C05459=1078.522,130.349,-70.098,174.153,23.499,154.054
C05460=1078.528,130.599,-70.117,174.156,23.501,154.054
C05461=1078.534,130.848,-70.137,174.158,23.504,154.054
C05462=1078.540,131.096,-70.157,174.159,23.506,154.055
C05463=1078.545,131.346,-70.177,174.162,23.509,154.055
C05464=1078.551,131.595,-70.197,174.163,23.510,154.055
C05465=1078.557,131.844,-70.217,174.165,23.513,154.055
C05466=1078.563,132.093,-70.236,174.167,23.515,154.056
C05467=1078.568,132.342,-70.257,174.169,23.517,154.056
C05468=1078.574,132.591,-70.277,174.170,23.520,154.056
C05469=1078.580,132.841,-70.296,174.173,23.522,154.056
C05470=1078.585,133.090,-70.317,174.174,23.524,154.056
C05471=1078.591,133.339,-70.337,174.176,23.527,154.057
C05472=1078.596,133.588,-70.357,174.178,23.529,154.057
C05473=1078.602,133.837,-70.376,174.180,23.532,154.057
C05474=1078.607,134.086,-70.397,174.181,23.533,154.057
C05475=1078.613,134.335,-70.417,174.184,23.536,154.058
C05476=1078.619,134.584,-70.437,174.186,23.538,154.058
C05477=1078.625,134.833,-70.457,174.187,23.541,154.058
C05478=1078.630,135.083,-70.478,174.190,23.543,154.058
C05479=1078.636,135.332,-70.498,174.191,23.545,154.058
C05480=1078.642,135.581,-70.518,174.193,23.548,154.058
C05481=1078.647,135.830,-70.538,174.195,23.550,154.059
C05482=1078.653,136.079,-70.558,174.197,23.552,154.059
C05483=1078.659,136.328,-70.579,174.198,23.555,154.059
C05484=1078.664,136.578,-70.598,174.201,23.557,154.059
C05485=1078.670,136.827,-70.618,174.203,23.559,154.059
C05486=1078.676,137.075,-70.638,174.204,23.561,154.060
C05487=1078.681,137.325,-70.659,174.207,23.564,154.060
C05488=1078.687,137.574,-70.679,174.208,23.566,154.060
C05489=1078.693,137.823,-70.700,174.210,23.568,154.060
C05490=1078.699,138.072,-70.720,174.212,23.571,154.061
C05491=1078.704,138.321,-70.740,174.214,23.573,154.061
C05492=1078.710,138.570,-70.760,174.215,23.575,154.061
C05493=1078.715,138.819,-70.781,174.218,23.577,154.061
C05494=1078.720,139.068,-70.801,174.220,23.580,154.061
C05495=1078.727,139.318,-70.822,174.221,23.582,154.062
C05496=1078.732,139.567,-70.842,174.224,23.584,154.062
C05497=1078.738,139.816,-70.862,174.225,23.587,154.062
C05498=1078.744,140.065,-70.883,174.228,23.589,154.062
C05499=1078.750,140.314,-70.903,174.229,23.591,154.063
C05500=1078.755,140.563,-70.923,174.231,23.594,154.063
C05501=1078.760,140.812,-70.944,174.233,23.596,154.063
C05502=1078.767,141.061,-70.964,174.235,23.598,154.063
C05503=1078.772,141.310,-70.985,174.237,23.601,154.063
C05504=1078.777,141.560,-71.005,174.239,23.603,154.064
C05505=1078.783,141.808,-71.025,174.241,23.605,154.064
C05506=1078.788,142.058,-71.046,174.243,23.608,154.064
C05507=1078.794,142.307,-71.066,174.244,23.610,154.064
C05508=1078.800,142.557,-71.087,174.247,23.612,154.064
C05509=1078.806,142.805,-71.107,174.248,23.615,154.065
C05510=1078.812,143.086,-71.131,174.251,23.617,154.065
C05511=1078.818,143.367,-71.154,174.253,23.620,154.065
C05512=1078.824,143.647,-71.176,174.255,23.622,154.065
C05513=1078.831,143.928,-71.200,174.257,23.625,154.066
C05514=1078.836,144.177,-71.221,174.260,23.627,154.066
C05515=1078.842,144.427,-71.242,174.261,23.629,154.066
C05516=1078.848,144.675,-71.262,174.263,23.632,154.066
C05517=1078.853,144.925,-71.282,174.265,23.634,154.066
C05518=1078.859,145.173,-71.303,174.267,23.637,154.067
C05519=1078.864,145.422,-71.324,174.269,23.639,154.067
C05520=1078.871,145.672,-71.344,174.271,23.641,154.067
C05521=1078.876,145.921,-71.365,174.273,23.643,154.067
C05522=1078.881,146.169,-71.386,174.274,23.645,154.067
C05523=1078.887,146.418,-71.407,174.277,23.648,154.068
C05524=1078.893,146.668,-71.427,174.279,23.650,154.068
C05525=1078.898,146.917,-71.448,174.281,23.652,154.068
C05526=1078.904,147.166,-71.469,174.283,23.655,154.068
C05527=1078.910,147.415,-71.490,174.285,23.657,154.068
C05528=1078.916,147.664,-71.510,174.286,23.659,154.069
C05529=1078.921,147.913,-71.530,174.289,23.662,154.069
C05530=1078.927,148.162,-71.552,174.290,23.663,154.069
C05531=1078.933,148.412,-71.572,174.293,23.666,154.069
C05532=1078.938,148.661,-71.593,174.295,23.668,154.069
C05533=1078.943,148.909,-71.614,174.296,23.671,154.070
C05534=1078.949,149.158,-71.635,174.299,23.673,154.070
C05535=1078.955,149.408,-71.655,174.301,23.675,154.070
C05536=1078.961,149.656,-71.676,174.302,23.677,154.070
C05537=1078.966,149.906,-71.697,174.305,23.680,154.070
C05538=1078.972,150.155,-71.719,174.306,23.682,154.071
C05539=1078.977,150.404,-71.739,174.308,23.684,154.071
C05540=1078.983,150.653,-71.760,174.311,23.687,154.071
C05541=1078.989,150.902,-71.781,174.312,23.689,154.071
C05542=1078.994,151.151,-71.802,174.314,23.691,154.071
C05543=1079.000,151.400,-71.823,174.317,23.694,154.072
C05544=1079.005,151.649,-71.844,174.318,23.696,154.072
C05545=1079.011,151.898,-71.865,174.321,23.698,154.072
C05546=1079.016,152.147,-71.886,174.323,23.701,154.072
C05547=1079.022,152.396,-71.907,174.324,23.702,154.072
C05548=1079.028,152.646,-71.928,174.326,23.705,154.073
C05549=1079.033,152.894,-71.949,174.328,23.707,154.073
C05550=1079.039,153.143,-71.970,174.330,23.709,154.073
C05551=1079.045,153.392,-71.992,174.333,23.712,154.073
C05552=1079.050,153.642,-72.012,174.334,23.714,154.073
C05553=1079.056,153.890,-72.033,174.336,23.716,154.073
C05554=1079.061,154.140,-72.054,174.339,23.719,154.074
C05555=1079.067,154.388,-72.076,174.340,23.721,154.074
C05556=1079.073,154.638,-72.096,174.342,23.723,154.074
C05557=1079.078,154.887,-72.118,174.345,23.726,154.074
C05558=1079.084,155.135,-72.139,174.346,23.727,154.074
C05559=1079.090,155.385,-72.160,174.349,23.730,154.075
C05560=1079.095,155.634,-72.181,174.351,23.732,154.075
C05561=1079.101,155.883,-72.202,174.352,23.734,154.075
C05562=1079.107,156.132,-72.223,174.354,23.737,154.075
C05563=1079.112,156.380,-72.245,174.357,23.739,154.075
C05564=1079.117,156.631,-72.266,174.358,23.741,154.076
C05565=1079.123,156.879,-72.287,174.361,23.744,154.076
C05566=1079.129,157.128,-72.309,174.363,23.746,154.076
C05567=1079.134,157.377,-72.330,174.364,23.748,154.076
C05568=1079.140,157.626,-72.351,174.367,23.751,154.076
C05569=1079.146,157.875,-72.373,174.369,23.753,154.077
C05570=1079.151,158.124,-72.393,174.371,23.755,154.077
C05571=1079.157,158.374,-72.415,174.373,23.757,154.077
C05572=1079.162,158.622,-72.437,174.375,23.760,154.077
C05573=1079.168,158.871,-72.458,174.377,23.762,154.077
C05574=1079.175,159.152,-72.482,174.380,23.764,154.078
C05575=1079.181,159.432,-72.506,174.382,23.767,154.078
C05576=1079.187,159.712,-72.529,174.384,23.769,154.078
C05577=1079.193,159.993,-72.554,174.387,23.772,154.078
C05578=1079.199,160.242,-72.575,174.388,23.774,154.078
C05579=1079.205,160.491,-72.597,174.390,23.777,154.079
C05580=1079.211,160.740,-72.618,174.393,23.779,154.079
C05581=1079.216,160.989,-72.639,174.395,23.781,154.079
C05582=1079.222,161.238,-72.661,174.396,23.784,154.079
C05583=1079.227,161.487,-72.682,174.399,23.786,154.079
C05584=1079.233,161.736,-72.704,174.401,23.788,154.080
C05585=1079.238,161.985,-72.726,174.402,23.790,154.080
C05586=1079.244,162.234,-72.747,174.405,23.793,154.080
C05587=1079.249,162.483,-72.769,174.407,23.795,154.080
C05588=1079.255,162.732,-72.791,174.409,23.797,154.080
C05589=1079.260,162.982,-72.812,174.411,23.800,154.081
C05590=1079.265,163.230,-72.833,174.413,23.802,154.081
C05591=1079.271,163.480,-72.855,174.415,23.805,154.081
C05592=1079.276,163.728,-72.877,174.417,23.807,154.081
C05593=1079.282,163.977,-72.898,174.419,23.809,154.081
C05594=1079.287,164.226,-72.920,174.422,23.812,154.082
C05595=1079.293,164.475,-72.942,174.424,23.814,154.082
C05596=1079.298,164.724,-72.964,174.425,23.816,154.082
C05597=1079.304,164.973,-72.985,174.428,23.818,154.082
C05598=1079.309,165.222,-73.007,174.430,23.821,154.082
C05599=1079.315,165.471,-73.029,174.432,23.823,154.083
C05600=1079.320,165.721,-73.051,174.434,23.825,154.083
C05601=1079.326,165.969,-73.072,174.436,23.828,154.083
C05602=1079.331,166.219,-73.094,174.438,23.830,154.083
C05603=1079.337,166.467,-73.116,174.440,23.832,154.083
C05604=1079.342,166.717,-73.138,174.442,23.835,154.084
C05605=1079.347,166.965,-73.160,174.444,23.837,154.084
C05606=1079.353,167.215,-73.181,174.447,23.840,154.084
C05607=1079.358,167.463,-73.203,174.448,23.841,154.084
C05608=1079.364,167.712,-73.226,174.450,23.844,154.084
C05609=1079.369,167.961,-73.248,174.453,23.846,154.085
C05610=1079.375,168.210,-73.269,174.455,23.848,154.085
C05611=1079.380,168.459,-73.291,174.457,23.851,154.085
C05612=1079.386,168.708,-73.313,174.459,23.853,154.085
C05613=1079.391,168.957,-73.335,174.461,23.855,154.085
C05614=1079.397,169.206,-73.356,174.464,23.858,154.086
C05615=1079.403,169.456,-73.378,174.466,23.860,154.086
C05616=1079.408,169.704,-73.401,174.467,23.863,154.086
C05617=1079.414,169.953,-73.423,174.470,23.865,154.086
C05618=1079.419,170.202,-73.444,174.472,23.867,154.086
C05619=1079.425,170.451,-73.466,174.474,23.870,154.087
C05620=1079.431,170.700,-73.488,174.476,23.871,154.087
C05621=1079.436,170.948,-73.510,174.478,23.874,154.087
C05622=1079.442,171.198,-73.533,174.480,23.876,154.087
C05623=1079.447,171.447,-73.554,174.483,23.879,154.087
C05624=1079.453,171.696,-73.576,174.484,23.880,154.087
C05625=1079.459,171.945,-73.599,174.487,23.883,154.088
C05626=1079.464,172.193,-73.620,174.489,23.885,154.088
C05627=1079.470,172.443,-73.642,174.491,23.888,154.088
C05628=1079.475,172.691,-73.665,174.494,23.890,154.088
C05629=1079.481,172.940,-73.687,174.495,23.892,154.088
C05630=1079.486,173.190,-73.709,174.497,23.894,154.089
C05631=1079.491,173.438,-73.732,174.500,23.897,154.089
C05632=1079.498,173.687,-73.753,174.502,23.899,154.089
C05633=1079.503,173.937,-73.775,174.504,23.901,154.089
C05634=1079.509,174.185,-73.797,174.506,23.903,154.089
C05635=1079.514,174.434,-73.820,174.508,23.905,154.089
C05636=1079.520,174.684,-73.842,174.511,23.908,154.090
C05637=1079.526,174.932,-73.864,174.513,23.910,154.090
C05638=1079.532,175.212,-73.889,174.515,23.913,154.090
C05639=1079.538,175.492,-73.914,174.518,23.915,154.090
C05640=1079.545,175.773,-73.939,174.520,23.918,154.091
C05641=1079.551,176.053,-73.964,174.522,23.920,154.091
C05642=1079.557,176.302,-73.987,174.525,23.922,154.091
C05643=1079.562,176.550,-74.008,174.527,23.925,154.091
C05644=1079.568,176.800,-74.031,174.529,23.927,154.091
C05645=1079.573,177.049,-74.054,174.532,23.930,154.091
C05646=1079.579,177.298,-74.075,174.533,23.931,154.092
C05647=1079.585,177.546,-74.098,174.535,23.934,154.092
C05648=1079.590,177.795,-74.120,174.538,23.936,154.092
C05649=1079.597,178.044,-74.142,174.540,23.939,154.092
C05650=1079.602,178.293,-74.165,174.543,23.941,154.092
C05651=1079.607,178.542,-74.187,174.545,23.943,154.092
C05652=1079.614,178.790,-74.209,174.546,23.945,154.093
C05653=1079.619,179.040,-74.232,174.549,23.947,154.093
C05654=1079.625,179.289,-74.255,174.551,23.950,154.093
C05655=1079.630,179.538,-74.277,174.554,23.952,154.093
C05656=1079.636,179.786,-74.299,174.556,23.955,154.093
C05657=1079.642,180.035,-74.322,174.558,23.957,154.093
C05658=1079.647,180.285,-74.344,174.560,23.959,154.094
C05659=1079.654,180.533,-74.366,174.562,23.961,154.094
C05660=1079.659,180.783,-74.389,174.564,23.963,154.094
C05661=1079.665,181.032,-74.412,174.567,23.966,154.094
C05662=1079.670,181.280,-74.434,174.569,23.968,154.094
C05663=1079.676,181.529,-74.456,174.571,23.970,154.094
C05664=1079.682,181.778,-74.479,174.574,23.972,154.095
C05665=1079.688,182.027,-74.502,174.575,23.974,154.095
C05666=1079.693,182.276,-74.524,174.578,23.976,154.095
C05667=1079.699,182.525,-74.546,174.580,23.979,154.095
C05668=1079.705,182.774,-74.569,174.582,23.981,154.095
C05669=1079.710,183.022,-74.592,174.585,23.983,154.095
C05670=1079.716,183.271,-74.614,174.587,23.986,154.096
C05671=1079.721,183.520,-74.637,174.590,23.988,154.096
C05672=1079.728,183.769,-74.659,174.592,23.990,154.096
C05673=1079.734,184.018,-74.682,174.594,23.992,154.096
C05674=1079.739,184.267,-74.704,174.596,23.995,154.096
C05675=1079.745,184.516,-74.727,174.598,23.997,154.096
C05676=1079.751,184.765,-74.750,174.601,23.999,154.097
C05677=1079.757,185.014,-74.773,174.603,24.001,154.097
C05678=1079.763,185.263,-74.796,174.605,24.003,154.097
C05679=1079.767,185.511,-74.819,174.608,24.006,154.097
C05680=1079.773,185.761,-74.841,174.610,24.008,154.097
C05681=1079.778,186.010,-74.864,174.611,24.011,154.098
C05682=1079.784,186.258,-74.887,174.614,24.013,154.098
C05683=1079.790,186.507,-74.910,174.616,24.015,154.098
C05684=1079.795,186.756,-74.932,174.618,24.018,154.098
C05685=1079.800,187.005,-74.956,174.621,24.020,154.098
C05686=1079.806,187.254,-74.979,174.623,24.023,154.099
C05687=1079.811,187.503,-75.002,174.625,24.025,154.099
C05688=1079.817,187.751,-75.025,174.628,24.027,154.099
C05689=1079.823,188.000,-75.048,174.630,24.030,154.099
C05690=1079.827,188.249,-75.071,174.633,24.032,154.099
C05691=1079.833,188.498,-75.094,174.634,24.034,154.099
C05692=1079.839,188.747,-75.117,174.636,24.036,154.100
C05693=1079.844,188.996,-75.140,174.639,24.039,154.100
C05694=1079.850,189.244,-75.163,174.641,24.041,154.100
C05695=1079.855,189.494,-75.186,174.643,24.044,154.100
C05696=1079.861,189.743,-75.209,174.646,24.046,154.100
C05697=1079.867,189.991,-75.232,174.648,24.048,154.101
C05698=1079.872,190.240,-75.255,174.650,24.051,154.101
C05699=1079.877,190.488,-75.278,174.653,24.053,154.101
C05700=1079.882,190.738,-75.301,174.655,24.055,154.101
C05701=1079.888,190.987,-75.324,174.657,24.058,154.101
C05702=1079.895,191.267,-75.350,174.660,24.060,154.102
C05703=1079.901,191.546,-75.376,174.662,24.063,154.102
C05704=1079.907,191.827,-75.403,174.665,24.066,154.102
C05705=1079.913,192.106,-75.429,174.668,24.068,154.102
C05706=1079.919,192.355,-75.452,174.670,24.070,154.102
C05707=1079.925,192.604,-75.474,174.672,24.073,154.103
C05708=1079.930,192.853,-75.498,174.675,24.075,154.103
C05709=1079.936,193.101,-75.522,174.677,24.077,154.103
C05710=1079.941,193.350,-75.545,174.679,24.080,154.103
C05711=1079.947,193.599,-75.568,174.681,24.082,154.103
C05712=1079.952,193.848,-75.591,174.683,24.084,154.103
C05713=1079.958,194.097,-75.614,174.686,24.087,154.104
C05714=1079.964,194.345,-75.638,174.688,24.089,154.104
C05715=1079.969,194.595,-75.661,174.690,24.091,154.104
C05716=1079.975,194.844,-75.684,174.693,24.093,154.104
C05717=1079.980,195.092,-75.707,174.695,24.096,154.104
C05718=1079.986,195.341,-75.731,174.697,24.098,154.105
C05719=1079.991,195.590,-75.754,174.700,24.100,154.105
C05720=1079.997,195.839,-75.777,174.702,24.103,154.105
C05721=1080.003,196.087,-75.801,174.704,24.105,154.105
C05722=1080.008,196.336,-75.825,174.707,24.107,154.105
C05723=1080.014,196.585,-75.847,174.709,24.110,154.105
C05724=1080.020,196.833,-75.871,174.712,24.112,154.106
C05725=1080.025,197.083,-75.895,174.714,24.114,154.106
C05726=1080.031,197.332,-75.918,174.716,24.117,154.106
C05727=1080.037,197.581,-75.942,174.719,24.119,154.106
C05728=1080.042,197.830,-75.965,174.721,24.121,154.106
C05729=1080.048,198.079,-75.988,174.723,24.124,154.107
C05730=1080.054,198.327,-76.012,174.726,24.126,154.107
C05731=1080.059,198.576,-76.035,174.728,24.128,154.107
C05732=1080.065,198.824,-76.059,174.731,24.131,154.107
C05733=1080.071,199.073,-76.082,174.733,24.133,154.107
C05734=1080.076,199.322,-76.106,174.735,24.135,154.107
C05735=1080.082,199.571,-76.129,174.738,24.137,154.108
C05736=1080.087,199.821,-76.153,174.740,24.140,154.108
C05737=1080.093,200.069,-76.177,174.742,24.142,154.108
C05738=1080.099,200.318,-76.200,174.745,24.144,154.108
C05739=1080.104,200.566,-76.224,174.747,24.147,154.108
C05740=1080.110,200.815,-76.247,174.749,24.149,154.108
C05741=1080.116,201.064,-76.271,174.752,24.151,154.109
C05742=1080.122,201.313,-76.295,174.754,24.154,154.109
C05743=1080.128,201.562,-76.318,174.757,24.156,154.109
C05744=1080.133,201.810,-76.342,174.759,24.159,154.109
C05745=1080.139,202.059,-76.365,174.761,24.161,154.109
C05746=1080.144,202.308,-76.390,174.764,24.163,154.109
C05747=1080.151,202.557,-76.413,174.766,24.165,154.110
C05748=1080.156,202.806,-76.437,174.768,24.168,154.110
C05749=1080.162,203.054,-76.461,174.771,24.170,154.110
C05750=1080.167,203.304,-76.484,174.773,24.172,154.110
C05751=1080.173,203.552,-76.508,174.776,24.175,154.110
C05752=1080.178,203.800,-76.532,174.778,24.177,154.111
C05753=1080.184,204.050,-76.556,174.780,24.179,154.111
C05754=1080.190,204.299,-76.580,174.783,24.182,154.111
C05755=1080.195,204.547,-76.604,174.785,24.184,154.111
C05756=1080.200,204.796,-76.628,174.787,24.186,154.111
C05757=1080.206,205.045,-76.651,174.791,24.189,154.112
C05758=1080.211,205.293,-76.676,174.793,24.192,154.112
C05759=1080.217,205.543,-76.700,174.795,24.194,154.112
C05760=1080.223,205.791,-76.723,174.798,24.196,154.112
C05761=1080.228,206.040,-76.747,174.800,24.199,154.112
C05762=1080.234,206.289,-76.772,174.803,24.201,154.112
C05763=1080.240,206.538,-76.796,174.805,24.203,154.113
C05764=1080.245,206.787,-76.819,174.807,24.206,154.113
C05765=1080.251,207.035,-76.843,174.809,24.208,154.113
C05766=1080.274,208.069,-76.943,174.909,24.261,154.111
C05767=1080.283,208.468,-76.983,174.913,24.267,154.112
C05768=1080.292,208.867,-77.022,174.917,24.272,154.113
C05769=1080.302,209.266,-77.061,174.921,24.277,154.113
C05770=1080.311,209.665,-77.101,174.924,24.282,154.114
C05771=1080.317,209.914,-77.126,174.926,24.286,154.114
C05772=1080.322,210.163,-77.150,174.929,24.289,154.115
C05773=1080.328,210.411,-77.175,174.931,24.293,154.115
C05774=1080.334,210.660,-77.200,174.934,24.296,154.116
C05775=1080.339,210.909,-77.224,174.936,24.299,154.116
C05776=1080.345,211.157,-77.249,174.938,24.303,154.116
C05777=1080.351,211.406,-77.274,174.940,24.306,154.117
C05778=1080.356,211.655,-77.298,174.943,24.309,154.117
C05779=1080.362,211.904,-77.323,174.945,24.313,154.118
C05780=1080.368,212.152,-77.348,174.947,24.316,154.118
C05781=1080.373,212.401,-77.374,174.949,24.319,154.118
C05782=1080.378,212.650,-77.398,174.952,24.323,154.119
C05783=1080.385,212.899,-77.423,174.954,24.326,154.119
C05784=1080.391,213.148,-77.448,174.957,24.329,154.120
C05785=1080.396,213.396,-77.472,174.959,24.332,154.120
C05786=1080.402,213.645,-77.497,174.961,24.336,154.121
C05787=1080.407,213.894,-77.522,174.964,24.340,154.121
C05788=1080.413,214.143,-77.548,174.966,24.343,154.121
C05789=1080.418,214.391,-77.573,174.968,24.346,154.122
C05790=1080.424,214.640,-77.597,174.970,24.349,154.122
C05791=1080.430,214.888,-77.622,174.973,24.353,154.122
C05792=1080.436,215.137,-77.647,174.975,24.356,154.123
C05793=1080.441,215.385,-77.672,174.977,24.359,154.123
C05794=1080.447,215.635,-77.697,174.979,24.362,154.124
C05795=1080.453,215.883,-77.722,174.982,24.366,154.124
C05796=1080.458,216.131,-77.747,174.984,24.370,154.125
C05797=1080.464,216.381,-77.772,174.986,24.373,154.125
C05798=1080.469,216.629,-77.797,174.989,24.376,154.125
C05799=1080.475,216.878,-77.822,174.992,24.380,154.126
C05800=1080.481,217.127,-77.847,174.994,24.383,154.126
C05801=1080.486,217.375,-77.873,174.996,24.386,154.127
C05802=1080.492,217.624,-77.898,174.998,24.389,154.127
C05803=1080.498,217.872,-77.923,175.001,24.393,154.127
C05804=1080.504,218.121,-77.948,175.003,24.396,154.128
C05805=1080.509,218.370,-77.974,175.005,24.399,154.128
C05806=1080.515,218.619,-77.998,175.007,24.402,154.129
C05807=1080.521,218.867,-78.023,175.010,24.406,154.129
C05808=1080.526,219.116,-78.049,175.013,24.409,154.129
C05809=1080.532,219.364,-78.074,175.015,24.412,154.130
C05810=1080.538,219.614,-78.099,175.018,24.416,154.130
C05811=1080.544,219.862,-78.124,175.020,24.420,154.131
C05812=1080.549,220.111,-78.150,175.022,24.423,154.131
C05813=1080.555,220.359,-78.175,175.024,24.426,154.132
C05814=1080.561,220.608,-78.201,175.027,24.430,154.132
C05815=1080.567,220.857,-78.226,175.029,24.433,154.132
C05816=1080.572,221.105,-78.251,175.031,24.436,154.133
C05817=1080.578,221.354,-78.276,175.033,24.439,154.133
C05818=1080.584,221.603,-78.302,175.036,24.443,154.133
C05819=1080.593,222.006,-78.343,175.040,24.448,154.134
C05820=1080.602,222.409,-78.385,175.044,24.453,154.135
C05821=1080.612,222.813,-78.426,175.048,24.459,154.135
C05822=1080.621,223.215,-78.467,175.052,24.464,154.136
C05823=1080.626,223.464,-78.493,175.054,24.467,154.136
C05824=1080.632,223.713,-78.518,175.057,24.471,154.137
C05825=1080.637,223.961,-78.544,175.059,24.474,154.137
C05826=1080.643,224.210,-78.569,175.061,24.478,154.138
C05827=1080.649,224.459,-78.595,175.064,24.481,154.138
C05828=1080.655,224.707,-78.621,175.066,24.484,154.139
C05829=1080.660,224.956,-78.646,175.068,24.488,154.139
C05830=1080.666,225.204,-78.672,175.071,24.491,154.139
C05831=1080.672,225.453,-78.697,175.073,24.494,154.140
C05832=1080.677,225.702,-78.723,175.075,24.498,154.140
C05833=1080.683,225.950,-78.748,175.078,24.501,154.141
C05834=1080.688,226.199,-78.774,175.081,24.504,154.141
C05835=1080.694,226.448,-78.800,175.083,24.508,154.142
C05836=1080.700,226.697,-78.826,175.085,24.511,154.142
C05837=1080.706,226.945,-78.852,175.088,24.515,154.142
C05838=1080.711,227.193,-78.877,175.090,24.518,154.143
C05839=1080.717,227.442,-78.903,175.092,24.521,154.143
C05840=1080.723,227.691,-78.928,175.095,24.525,154.143
C05841=1080.728,227.940,-78.954,175.097,24.528,154.144
C05842=1080.735,228.188,-78.980,175.099,24.531,154.144
C05843=1080.740,228.437,-79.006,175.102,24.535,154.145
C05844=1080.746,228.686,-79.032,175.105,24.538,154.145
C05845=1080.751,228.934,-79.057,175.107,24.541,154.145
C05846=1080.757,229.182,-79.084,175.110,24.545,154.146
C05847=1080.763,229.431,-79.110,175.112,24.548,154.146
C05848=1080.769,229.680,-79.135,175.114,24.551,154.147
C05849=1080.774,229.929,-79.161,175.117,24.554,154.147
C05850=1080.780,230.177,-79.188,175.119,24.558,154.147
C05851=1080.786,230.426,-79.213,175.121,24.561,154.148
C05852=1080.792,230.675,-79.239,175.124,24.564,154.148
C05853=1080.797,230.922,-79.265,175.127,24.568,154.149
C05854=1080.802,231.171,-79.291,175.129,24.571,154.149
C05855=1080.809,231.420,-79.317,175.132,24.575,154.150
C05856=1080.814,231.668,-79.343,175.134,24.578,154.150
C05857=1080.820,231.917,-79.369,175.136,24.581,154.150
C05858=1080.826,232.166,-79.396,175.139,24.585,154.151
C05859=1080.831,232.415,-79.422,175.141,24.588,154.151
C05860=1080.837,232.663,-79.448,175.143,24.591,154.152
C05861=1080.843,232.912,-79.474,175.146,24.595,154.152
C05862=1080.849,233.160,-79.500,175.148,24.598,154.152
C05863=1080.854,233.409,-79.526,175.151,24.601,154.153
C05864=1080.859,233.657,-79.552,175.154,24.605,154.153
C05865=1080.865,233.906,-79.579,175.156,24.608,154.154
C05866=1080.871,234.154,-79.605,175.159,24.612,154.154
C05867=1080.876,234.403,-79.631,175.161,24.615,154.154
C05868=1080.882,234.651,-79.658,175.163,24.618,154.155
C05869=1080.888,234.900,-79.683,175.166,24.622,154.155
C05870=1080.894,235.148,-79.710,175.168,24.625,154.156
C05871=1080.903,235.543,-79.752,175.172,24.630,154.156
C05872=1080.911,235.938,-79.793,175.176,24.636,154.157
C05873=1080.921,236.333,-79.835,175.180,24.641,154.158
C05874=1080.930,236.728,-79.878,175.184,24.646,154.158
C05875=1080.935,236.976,-79.904,175.187,24.650,154.159
C05876=1080.941,237.225,-79.930,175.189,24.653,154.159
C05877=1080.947,237.474,-79.957,175.192,24.657,154.160
C05878=1080.952,237.722,-79.983,175.194,24.660,154.160
C05879=1080.958,237.971,-80.009,175.196,24.663,154.160
C05880=1080.964,238.219,-80.036,175.199,24.667,154.161
C05881=1080.969,238.468,-80.063,175.201,24.670,154.161
C05882=1080.975,238.716,-80.089,175.204,24.673,154.162
C05883=1080.981,238.965,-80.115,175.206,24.677,154.162
C05884=1080.986,239.213,-80.142,175.209,24.680,154.162
C05885=1080.992,239.462,-80.169,175.212,24.683,154.163
C05886=1080.998,239.710,-80.195,175.214,24.686,154.163
C05887=1081.004,239.958,-80.222,175.217,24.690,154.164
C05888=1081.009,240.207,-80.248,175.219,24.694,154.164
C05889=1081.016,240.456,-80.275,175.221,24.697,154.165
C05890=1081.021,240.705,-80.301,175.224,24.700,154.165
C05891=1081.027,240.953,-80.328,175.226,24.704,154.165
C05892=1081.033,241.201,-80.355,175.229,24.707,154.166
C05893=1081.038,241.450,-80.382,175.231,24.710,154.166
C05894=1081.044,241.698,-80.409,175.234,24.714,154.166
C05895=1081.050,241.947,-80.435,175.237,24.717,154.167
C05896=1081.055,242.195,-80.462,175.239,24.720,154.167
C05897=1081.061,242.444,-80.489,175.242,24.724,154.168
C05898=1081.067,242.693,-80.516,175.244,24.727,154.168
C05899=1081.073,242.941,-80.542,175.247,24.730,154.168
C05900=1081.078,243.190,-80.569,175.249,24.734,154.169
C05901=1081.084,243.438,-80.596,175.252,24.738,154.169
C05902=1081.090,243.686,-80.623,175.254,24.741,154.170
C05903=1081.096,243.935,-80.649,175.256,24.744,154.170
C05904=1081.101,244.183,-80.677,175.260,24.747,154.171
C05905=1081.106,244.432,-80.703,175.262,24.751,154.171
C05906=1081.113,244.681,-80.730,175.265,24.755,154.172
C05907=1081.118,244.930,-80.758,175.267,24.758,154.172
C05908=1081.124,245.178,-80.784,175.270,24.761,154.172
C05909=1081.129,245.426,-80.811,175.272,24.764,154.173
C05910=1081.134,245.675,-80.838,175.274,24.768,154.173
C05911=1081.140,245.923,-80.865,175.277,24.771,154.174
C05912=1081.147,246.172,-80.892,175.279,24.775,154.174
C05913=1081.152,246.420,-80.920,175.282,24.778,154.174
C05914=1081.158,246.669,-80.946,175.284,24.781,154.175
C05915=1081.163,246.917,-80.973,175.288,24.785,154.175
C05916=1081.168,247.166,-81.000,175.290,24.788,154.176
C05917=1081.175,247.413,-81.028,175.293,24.792,154.176
C05918=1081.180,247.663,-81.055,175.295,24.795,154.177
C05919=1081.186,247.911,-81.082,175.297,24.799,154.177
C05920=1081.191,248.160,-81.109,175.300,24.802,154.177
C05921=1081.197,248.408,-81.136,175.302,24.805,154.178
C05922=1081.202,248.656,-81.164,175.305,24.809,154.178
C05923=1081.211,249.044,-81.206,175.309,24.814,154.179
C05924=1081.220,249.432,-81.248,175.313,24.820,154.180
C05925=1081.228,249.820,-81.291,175.317,24.825,154.180
C05926=1081.238,250.208,-81.334,175.321,24.830,154.181
C05927=1081.243,250.457,-81.361,175.324,24.834,154.181
C05928=1081.249,250.705,-81.389,175.326,24.837,154.182
C05929=1081.254,250.954,-81.416,175.329,24.841,154.182
C05930=1081.260,251.201,-81.443,175.331,24.844,154.183
C05931=1081.266,251.451,-81.471,175.334,24.848,154.183
C05932=1081.271,251.700,-81.498,175.336,24.851,154.184
C05933=1081.277,251.947,-81.526,175.339,24.855,154.184
C05934=1081.282,252.196,-81.553,175.341,24.858,154.184
C05935=1081.289,252.444,-81.581,175.344,24.862,154.185
C05936=1081.294,252.693,-81.608,175.347,24.865,154.185
C05937=1081.299,252.941,-81.636,175.350,24.869,154.186
C05938=1081.306,253.190,-81.663,175.352,24.872,154.186
C05939=1081.311,253.438,-81.691,175.355,24.875,154.186
C05940=1081.317,253.686,-81.718,175.357,24.878,154.187
C05941=1081.323,253.935,-81.746,175.360,24.883,154.187
C05942=1081.328,254.183,-81.774,175.362,24.886,154.188
C05943=1081.334,254.432,-81.800,175.365,24.889,154.188
C05944=1081.340,254.681,-81.829,175.367,24.892,154.189
C05945=1081.345,254.929,-81.857,175.370,24.896,154.189
C05946=1081.351,255.177,-81.883,175.373,24.899,154.189
C05947=1081.357,255.426,-81.912,175.376,24.903,154.190
C05948=1081.363,255.673,-81.939,175.378,24.906,154.190
C05949=1081.368,255.922,-81.966,175.381,24.910,154.191
C05950=1081.374,256.171,-81.995,175.383,24.913,154.191
C05951=1081.380,256.419,-82.022,175.386,24.916,154.191
C05952=1081.386,256.668,-82.050,175.388,24.920,154.192
C05953=1081.391,256.916,-82.078,175.391,24.923,154.192
C05954=1081.397,257.164,-82.105,175.393,24.927,154.193
C05955=1081.403,257.412,-82.133,175.396,24.930,154.193
C05956=1081.408,257.661,-82.160,175.399,24.933,154.194
C05957=1081.414,257.910,-82.189,175.402,24.937,154.194
C05958=1081.420,258.158,-82.216,175.404,24.940,154.195
C05959=1081.426,258.406,-82.244,175.407,24.944,154.195
C05960=1081.431,258.654,-82.272,175.409,24.947,154.195
C05961=1081.438,258.903,-82.300,175.412,24.951,154.196
C05962=1081.443,259.152,-82.327,175.415,24.954,154.196
C05963=1081.449,259.400,-82.356,175.417,24.957,154.197
C05964=1081.454,259.648,-82.384,175.420,24.961,154.197
C05965=1081.461,259.897,-82.411,175.423,24.964,154.197
C05966=1081.466,260.145,-82.439,175.426,24.968,154.198
C05967=1081.472,260.394,-82.468,175.428,24.971,154.198
C05968=1081.478,260.642,-82.496,175.431,24.975,154.199
C05969=1081.484,260.890,-82.523,175.433,24.978,154.199
C05970=1081.490,261.138,-82.551,175.436,24.982,154.200
C05971=1081.496,261.387,-82.580,175.438,24.985,154.200
C05972=1081.501,261.635,-82.608,175.441,24.988,154.200
C05973=1081.508,261.883,-82.635,175.444,24.992,154.201
C05974=1081.513,262.131,-82.663,175.447,24.995,154.201
C05975=1081.522,262.517,-82.707,175.451,25.001,154.202
C05976=1081.531,262.903,-82.751,175.455,25.006,154.202
C05977=1081.540,263.287,-82.795,175.459,25.011,154.203
C05978=1081.550,263.673,-82.838,175.463,25.016,154.204
C05979=1081.556,263.921,-82.866,175.466,25.020,154.204
C05980=1081.561,264.169,-82.894,175.468,25.023,154.205
C05981=1081.567,264.418,-82.922,175.471,25.026,154.205
C05982=1081.573,264.666,-82.951,175.474,25.030,154.206
C05983=1081.579,264.914,-82.979,175.477,25.034,154.206
C05984=1081.584,265.162,-83.007,175.480,25.037,154.206
C05985=1081.590,265.411,-83.036,175.482,25.041,154.207
C05986=1081.596,265.659,-83.064,175.485,25.044,154.207
C05987=1081.602,265.907,-83.093,175.487,25.047,154.208
C05988=1081.607,266.156,-83.121,175.490,25.051,154.208
C05989=1081.612,266.404,-83.149,175.492,25.054,154.209
C05990=1081.618,266.653,-83.178,175.495,25.058,154.209
C05991=1081.624,266.901,-83.206,175.498,25.062,154.209
C05992=1081.630,267.149,-83.235,175.500,25.065,154.210
C05993=1081.636,267.398,-83.264,175.504,25.069,154.210
C05994=1081.641,267.646,-83.292,175.506,25.072,154.211
C05995=1081.647,267.894,-83.320,175.509,25.076,154.211
C05996=1081.653,268.142,-83.349,175.512,25.079,154.212
C05997=1081.659,268.390,-83.377,175.514,25.083,154.212
C05998=1081.665,268.639,-83.405,175.517,25.086,154.213
C05999=1081.670,268.887,-83.435,175.519,25.089,154.213
C06000=1081.676,269.136,-83.463,175.522,25.093,154.213
C06001=1081.682,269.384,-83.492,175.525,25.097,154.214
C06002=1081.687,269.632,-83.520,175.527,25.100,154.214
C06003=1081.693,269.880,-83.549,175.531,25.103,154.215
C06004=1081.699,270.129,-83.577,175.533,25.107,154.215
C06005=1081.704,270.377,-83.607,175.536,25.111,154.216
C06006=1081.710,270.625,-83.635,175.539,25.115,154.216
C06007=1081.716,270.873,-83.664,175.541,25.118,154.217
C06008=1081.722,271.121,-83.692,175.544,25.121,154.217
C06009=1081.727,271.370,-83.722,175.546,25.125,154.217
C06010=1081.733,271.619,-83.750,175.549,25.128,154.218
C06011=1081.739,271.867,-83.779,175.552,25.132,154.218
C06012=1081.745,272.115,-83.807,175.554,25.135,154.219
C06013=1081.750,272.363,-83.837,175.558,25.139,154.219
C06014=1081.757,272.611,-83.866,175.561,25.142,154.220
C06015=1081.762,272.859,-83.894,175.563,25.146,154.220
C06016=1081.767,273.108,-83.923,175.566,25.149,154.220
C06017=1081.774,273.356,-83.952,175.568,25.153,154.221
C06018=1081.780,273.605,-83.981,175.571,25.157,154.221
C06019=1081.785,273.853,-84.010,175.574,25.160,154.222
C06020=1081.791,274.101,-84.039,175.576,25.164,154.222
C06021=1081.797,274.349,-84.068,175.579,25.167,154.223
C06022=1081.802,274.598,-84.097,175.582,25.171,154.223
C06023=1081.808,274.845,-84.125,175.584,25.174,154.224
C06024=1081.813,275.094,-84.155,175.587,25.178,154.224
C06025=1081.820,275.342,-84.184,175.591,25.182,154.225
C06026=1081.826,275.591,-84.212,175.593,25.185,154.225
C06027=1081.834,275.978,-84.258,175.597,25.191,154.226
C06028=1081.843,276.366,-84.304,175.602,25.196,154.226
C06029=1081.853,276.755,-84.350,175.605,25.202,154.227
C06030=1081.860,277.143,-84.395,175.610,25.207,154.228
C06031=1081.867,277.391,-84.424,175.613,25.211,154.228
C06032=1081.872,277.640,-84.454,175.615,25.214,154.229
C06033=1081.879,277.888,-84.483,175.618,25.218,154.229
C06034=1081.883,278.136,-84.512,175.621,25.222,154.230
C06035=1081.890,278.384,-84.541,175.623,25.226,154.230
C06036=1081.895,278.632,-84.571,175.627,25.229,154.231
C06037=1081.901,278.881,-84.600,175.630,25.233,154.231
C06038=1081.907,279.129,-84.629,175.632,25.236,154.232
C06039=1081.913,279.377,-84.658,175.635,25.240,154.232
C06040=1081.919,279.626,-84.688,175.638,25.244,154.233
C06041=1081.924,279.873,-84.717,175.640,25.247,154.233
C06042=1081.930,280.121,-84.746,175.643,25.251,154.233
C06043=1081.935,280.370,-84.776,175.646,25.255,154.234
C06044=1081.942,280.618,-84.805,175.648,25.258,154.234
C06045=1081.947,280.866,-84.835,175.651,25.261,154.235
C06046=1081.954,281.114,-84.864,175.654,25.265,154.235
C06047=1081.959,281.362,-84.894,175.656,25.269,154.236
C06048=1081.965,281.611,-84.924,175.660,25.272,154.236
C06049=1081.971,281.859,-84.953,175.663,25.276,154.237
C06050=1081.976,282.107,-84.982,175.665,25.279,154.237
C06051=1081.982,282.354,-85.012,175.668,25.283,154.238
C06052=1081.987,282.603,-85.042,175.671,25.287,154.238
C06053=1081.993,282.851,-85.071,175.674,25.291,154.239
C06054=1081.999,283.100,-85.101,175.676,25.294,154.239
C06055=1082.004,283.348,-85.130,175.679,25.298,154.240
C06056=1082.010,283.596,-85.161,175.682,25.302,154.240
C06057=1082.017,283.844,-85.190,175.684,25.305,154.241
C06058=1082.022,284.092,-85.219,175.687,25.309,154.241
C06059=1082.028,284.340,-85.250,175.690,25.313,154.242
C06060=1082.033,284.589,-85.279,175.693,25.316,154.242
C06061=1082.039,284.837,-85.309,175.696,25.320,154.242
C06062=1082.045,285.085,-85.339,175.699,25.324,154.243
C06063=1082.051,285.333,-85.368,175.702,25.327,154.243
C06064=1082.056,285.581,-85.398,175.704,25.331,154.244
C06065=1082.062,285.829,-85.428,175.707,25.335,154.244
C06066=1082.068,286.078,-85.458,175.710,25.338,154.245
C06067=1082.074,286.325,-85.488,175.713,25.342,154.245
C06068=1082.080,286.574,-85.517,175.715,25.345,154.246
C06069=1082.086,286.821,-85.548,175.718,25.349,154.246
C06070=1082.091,287.070,-85.577,175.721,25.353,154.247
C06071=1082.097,287.318,-85.608,175.723,25.356,154.247
C06072=1082.103,287.566,-85.637,175.726,25.360,154.248
C06073=1082.109,287.814,-85.667,175.729,25.364,154.248
C06074=1082.115,288.062,-85.697,175.732,25.368,154.249
C06075=1082.120,288.310,-85.727,175.735,25.371,154.249
C06076=1082.126,288.558,-85.757,175.738,25.375,154.250
C06077=1082.132,288.806,-85.787,175.741,25.379,154.250
C06078=1082.137,289.055,-85.817,175.744,25.383,154.251
C06079=1082.147,289.453,-85.865,175.748,25.388,154.251
C06080=1082.156,289.850,-85.914,175.753,25.395,154.252
C06081=1082.166,290.248,-85.962,175.757,25.400,154.253
C06082=1082.174,290.646,-86.010,175.762,25.406,154.254
C06083=1082.180,290.894,-86.040,175.764,25.410,154.254
C06084=1082.186,291.142,-86.071,175.767,25.413,154.255
C06085=1082.192,291.390,-86.100,175.770,25.417,154.255
C06086=1082.198,291.639,-86.131,175.773,25.421,154.256
C06087=1082.204,291.887,-86.161,175.776,25.425,154.256
C06088=1082.210,292.135,-86.192,175.778,25.428,154.257
C06089=1082.215,292.382,-86.222,175.781,25.432,154.257
C06090=1082.221,292.631,-86.252,175.784,25.436,154.258
C06091=1082.227,292.879,-86.282,175.787,25.440,154.258
C06092=1082.233,293.126,-86.312,175.790,25.443,154.259
C06093=1082.238,293.374,-86.343,175.793,25.447,154.259
C06094=1082.244,293.623,-86.374,175.796,25.451,154.260
C06095=1082.250,293.871,-86.404,175.799,25.455,154.260
C06096=1082.256,294.119,-86.435,175.802,25.459,154.261
C06097=1082.261,294.367,-86.464,175.804,25.463,154.261
C06098=1082.267,294.615,-86.495,175.807,25.466,154.262
C06099=1082.273,294.863,-86.525,175.810,25.470,154.262
C06100=1082.279,295.111,-86.556,175.813,25.474,154.263
C06101=1082.285,295.359,-86.586,175.816,25.478,154.263
C06102=1082.290,295.607,-86.617,175.818,25.482,154.264
C06103=1082.296,295.855,-86.647,175.821,25.485,154.264
C06104=1082.302,296.103,-86.678,175.824,25.489,154.265
C06105=1082.308,296.351,-86.708,175.827,25.493,154.265
C06106=1082.313,296.600,-86.739,175.830,25.497,154.266
C06107=1082.319,296.847,-86.770,175.832,25.500,154.266
C06108=1082.325,297.095,-86.801,175.835,25.504,154.267
C06109=1082.332,297.343,-86.832,175.838,25.508,154.267
C06110=1082.337,297.591,-86.862,175.841,25.512,154.268
C06111=1082.343,297.839,-86.893,175.844,25.516,154.268
C06112=1082.348,298.087,-86.923,175.847,25.520,154.269
C06113=1082.354,298.336,-86.955,175.850,25.524,154.270
C06114=1082.360,298.584,-86.985,175.853,25.528,154.270
C06115=1082.365,298.831,-87.017,175.856,25.532,154.271
C06116=1082.371,299.079,-87.047,175.859,25.536,154.271
C06117=1082.376,299.327,-87.078,175.862,25.539,154.272
C06118=1082.383,299.576,-87.109,175.864,25.543,154.272
C06119=1082.388,299.823,-87.140,175.867,25.547,154.273
C06120=1082.394,300.071,-87.171,175.870,25.551,154.273
C06121=1082.399,300.319,-87.201,175.873,25.555,154.274
C06122=1082.405,300.567,-87.232,175.876,25.559,154.274
C06123=1082.411,300.815,-87.264,175.879,25.563,154.275
C06124=1082.417,301.063,-87.294,175.881,25.567,154.276
C06125=1082.422,301.311,-87.325,175.884,25.571,154.276
C06126=1082.428,301.559,-87.357,175.887,25.575,154.277
C06127=1082.433,301.807,-87.388,175.890,25.579,154.277
C06128=1082.440,302.054,-87.419,175.893,25.582,154.278
C06129=1082.445,302.302,-87.450,175.896,25.586,154.278
C06130=1082.451,302.551,-87.480,175.899,25.590,154.279
C06131=1082.461,302.963,-87.533,175.904,25.597,154.280
C06132=1082.470,303.375,-87.584,175.908,25.603,154.280
C06133=1082.479,303.787,-87.636,175.913,25.610,154.281
C06134=1082.489,304.199,-87.688,175.918,25.616,154.282
C06135=1082.494,304.447,-87.719,175.921,25.621,154.283
C06136=1082.501,304.695,-87.750,175.924,25.625,154.283
C06137=1082.506,304.943,-87.782,175.927,25.629,154.284
C06138=1082.512,305.191,-87.812,175.930,25.632,154.285
C06139=1082.518,305.439,-87.844,175.933,25.636,154.285
C06140=1082.523,305.687,-87.875,175.936,25.640,154.286
C06141=1082.530,305.935,-87.907,175.939,25.644,154.286
C06142=1082.535,306.182,-87.938,175.941,25.648,154.287
C06143=1082.541,306.431,-87.969,175.944,25.652,154.287
C06144=1082.547,306.678,-88.001,175.947,25.656,154.288
C06145=1082.552,306.926,-88.032,175.950,25.660,154.288
C06146=1082.559,307.174,-88.063,175.953,25.664,154.289
C06147=1082.564,307.422,-88.095,175.956,25.668,154.290
C06148=1082.570,307.670,-88.127,175.959,25.672,154.290
C06149=1082.576,307.917,-88.158,175.962,25.676,154.291
C06150=1082.582,308.166,-88.189,175.965,25.680,154.291
C06151=1082.587,308.414,-88.221,175.968,25.684,154.292
C06152=1082.594,308.662,-88.252,175.970,25.688,154.292
C06153=1082.599,308.909,-88.284,175.973,25.692,154.293
C06154=1082.605,309.157,-88.316,175.976,25.696,154.293
C06155=1082.611,309.405,-88.346,175.979,25.700,154.294
C06156=1082.617,309.653,-88.378,175.982,25.704,154.294
C06157=1082.623,309.902,-88.410,175.985,25.708,154.295
C06158=1082.629,310.149,-88.442,175.988,25.712,154.296
C06159=1082.635,310.397,-88.474,175.991,25.716,154.296
C06160=1082.641,310.644,-88.505,175.994,25.720,154.297
C06161=1082.647,310.893,-88.537,175.997,25.724,154.297
C06162=1082.653,311.140,-88.568,176.000,25.728,154.298
C06163=1082.659,311.388,-88.600,176.003,25.732,154.298
C06164=1082.665,311.636,-88.632,176.007,25.736,154.299
C06165=1082.670,311.884,-88.664,176.009,25.740,154.300
C06166=1082.677,312.132,-88.695,176.012,25.744,154.300
C06167=1082.683,312.380,-88.727,176.015,25.748,154.301
C06168=1082.688,312.627,-88.759,176.018,25.752,154.301
C06169=1082.694,312.876,-88.791,176.021,25.756,154.302
C06170=1082.700,313.124,-88.823,176.024,25.760,154.302
C06171=1082.706,313.371,-88.854,176.027,25.764,154.303
C06172=1082.712,313.619,-88.886,176.030,25.768,154.304
C06173=1082.718,313.867,-88.918,176.033,25.772,154.304
C06174=1082.724,314.115,-88.950,176.036,25.776,154.305
C06175=1082.730,314.363,-88.982,176.039,25.781,154.305
C06176=1082.737,314.610,-89.014,176.042,25.785,154.306
C06177=1082.743,314.859,-89.046,176.045,25.788,154.306
C06178=1082.748,315.106,-89.078,176.048,25.793,154.307
C06179=1082.753,315.355,-89.110,176.051,25.797,154.308
C06180=1082.759,315.602,-89.142,176.054,25.801,154.308
C06181=1082.765,315.850,-89.175,176.057,25.805,154.309
C06182=1082.771,316.098,-89.207,176.060,25.810,154.309
C06183=1082.781,316.513,-89.261,176.064,25.816,154.310
C06184=1082.790,316.928,-89.315,176.069,25.824,154.312
C06185=1082.799,317.344,-89.369,176.075,25.831,154.313
C06186=1082.809,317.759,-89.423,176.079,25.838,154.314
C06187=1082.814,318.006,-89.455,176.082,25.842,154.314
C06188=1082.820,318.254,-89.487,176.085,25.846,154.315
C06189=1082.826,318.502,-89.519,176.088,25.851,154.315
C06190=1082.832,318.750,-89.553,176.091,25.855,154.316
C06191=1082.837,318.998,-89.584,176.094,25.859,154.317
C06192=1082.844,319.245,-89.617,176.097,25.863,154.317
C06193=1082.849,319.494,-89.650,176.100,25.868,154.318
C06194=1082.855,319.741,-89.682,176.103,25.872,154.319
C06195=1082.861,319.989,-89.714,176.106,25.876,154.319
C06196=1082.867,320.236,-89.747,176.109,25.880,154.320
C06197=1082.872,320.485,-89.779,176.112,25.885,154.321
C06198=1082.878,320.733,-89.812,176.115,25.889,154.321
C06199=1082.884,320.980,-89.844,176.118,25.894,154.322
C06200=1082.889,321.228,-89.877,176.121,25.897,154.322
C06201=1082.896,321.476,-89.910,176.124,25.902,154.323
C06202=1082.902,321.724,-89.942,176.127,25.906,154.324
C06203=1082.907,321.972,-89.975,176.129,25.911,154.324
C06204=1082.913,322.219,-90.007,176.132,25.915,154.325
C06205=1082.919,322.467,-90.040,176.136,25.919,154.326
C06206=1082.924,322.715,-90.073,176.138,25.923,154.326
C06207=1082.931,322.962,-90.106,176.142,25.928,154.327
C06208=1082.937,323.211,-90.138,176.145,25.932,154.327
C06209=1082.942,323.458,-90.171,176.148,25.937,154.328
C06210=1082.949,323.706,-90.204,176.151,25.941,154.329
C06211=1082.955,323.954,-90.236,176.154,25.945,154.329
C06212=1082.959,324.201,-90.269,176.157,25.949,154.330
C06213=1082.966,324.449,-90.302,176.160,25.954,154.331
C06214=1082.972,324.697,-90.334,176.163,25.958,154.331
C06215=1082.978,324.945,-90.368,176.166,25.962,154.332
C06216=1082.984,325.193,-90.400,176.169,25.967,154.333
C06217=1082.989,325.441,-90.433,176.172,25.971,154.333
C06218=1082.995,325.688,-90.466,176.175,25.976,154.334
C06219=1083.002,325.936,-90.499,176.178,25.980,154.335
C06220=1083.007,326.184,-90.532,176.181,25.984,154.335
C06221=1083.014,326.431,-90.565,176.184,25.989,154.336
C06222=1083.019,326.679,-90.598,176.187,25.993,154.337
C06223=1083.025,326.927,-90.631,176.190,25.997,154.337
C06224=1083.031,327.175,-90.664,176.194,26.002,154.338
C06225=1083.037,327.422,-90.697,176.197,26.006,154.339
C06226=1083.044,327.670,-90.730,176.200,26.011,154.339
C06227=1083.049,327.918,-90.763,176.203,26.015,154.340
C06228=1083.055,328.165,-90.796,176.206,26.020,154.341
C06229=1083.061,328.413,-90.829,176.209,26.024,154.341
C06230=1083.067,328.661,-90.862,176.212,26.028,154.342
C06231=1083.073,328.909,-90.895,176.215,26.033,154.343
C06232=1083.079,329.156,-90.928,176.217,26.037,154.343
C06233=1083.085,329.405,-90.962,176.220,26.041,154.344
C06234=1083.092,329.653,-90.994,176.223,26.046,154.344
C06235=1083.101,330.060,-91.049,176.229,26.053,154.346
C06236=1083.111,330.469,-91.104,176.234,26.061,154.347
C06237=1083.121,330.878,-91.159,176.239,26.068,154.348
C06238=1083.131,331.286,-91.214,176.244,26.075,154.349
C06239=1083.137,331.534,-91.247,176.247,26.080,154.350
C06240=1083.143,331.781,-91.280,176.250,26.084,154.350
C06241=1083.149,332.029,-91.314,176.253,26.089,154.351
C06242=1083.154,332.277,-91.347,176.256,26.093,154.352
C06243=1083.160,332.524,-91.381,176.259,26.098,154.352
C06244=1083.167,332.772,-91.414,176.262,26.102,154.353
C06245=1083.172,333.020,-91.447,176.266,26.107,154.354
C06246=1083.179,333.268,-91.482,176.269,26.111,154.354
C06247=1083.184,333.516,-91.515,176.272,26.116,154.355
C06248=1083.190,333.764,-91.548,176.275,26.121,154.356
C06249=1083.196,334.011,-91.582,176.278,26.125,154.357
C06250=1083.202,334.259,-91.615,176.281,26.130,154.357
C06251=1083.208,334.506,-91.649,176.284,26.135,154.358
C06252=1083.213,334.754,-91.683,176.287,26.139,154.359
C06253=1083.220,335.002,-91.717,176.290,26.144,154.360
C06254=1083.225,335.250,-91.750,176.293,26.149,154.360
C06255=1083.231,335.497,-91.784,176.296,26.153,154.361
C06256=1083.238,335.744,-91.817,176.299,26.158,154.362
C06257=1083.243,335.992,-91.851,176.303,26.163,154.362
C06258=1083.250,336.240,-91.885,176.306,26.167,154.363
C06259=1083.255,336.488,-91.919,176.309,26.172,154.364
C06260=1083.261,336.735,-91.953,176.312,26.176,154.365
C06261=1083.267,336.983,-91.986,176.315,26.181,154.365
C06262=1083.273,337.230,-92.020,176.318,26.186,154.366
C06263=1083.279,337.478,-92.055,176.321,26.191,154.367
C06264=1083.285,337.726,-92.088,176.324,26.195,154.367
C06265=1083.291,337.973,-92.122,176.327,26.200,154.368
C06266=1083.298,338.221,-92.156,176.330,26.205,154.369
C06267=1083.303,338.469,-92.189,176.333,26.209,154.370
C06268=1083.308,338.716,-92.224,176.337,26.214,154.370
C06269=1083.314,338.964,-92.258,176.340,26.219,154.371
C06270=1083.321,339.212,-92.292,176.343,26.224,154.372
C06271=1083.326,339.460,-92.326,176.346,26.228,154.373
C06272=1083.332,339.707,-92.360,176.350,26.233,154.373
C06273=1083.338,339.954,-92.394,176.352,26.238,154.374
C06274=1083.344,340.202,-92.428,176.355,26.243,154.375
C06275=1083.350,340.449,-92.462,176.358,26.248,154.376
C06276=1083.356,340.697,-92.496,176.361,26.252,154.376
C06277=1083.363,340.945,-92.531,176.365,26.257,154.377
C06278=1083.368,341.192,-92.565,176.368,26.262,154.378
C06279=1083.373,341.440,-92.599,176.371,26.267,154.379
C06280=1083.380,341.688,-92.633,176.374,26.272,154.380
C06281=1083.386,341.936,-92.667,176.378,26.277,154.380
C06282=1083.392,342.183,-92.701,176.380,26.282,154.381
C06283=1083.398,342.431,-92.736,176.383,26.287,154.382
C06284=1083.404,342.678,-92.770,176.386,26.292,154.383
C06285=1083.409,342.926,-92.804,176.390,26.297,154.384
C06286=1083.416,343.173,-92.840,176.393,26.301,154.384
C06287=1083.426,343.576,-92.895,176.398,26.309,154.386
C06288=1083.435,343.979,-92.951,176.403,26.317,154.387
C06289=1083.444,344.382,-93.007,176.408,26.325,154.388
C06290=1083.455,344.784,-93.063,176.414,26.333,154.389
C06291=1083.461,345.032,-93.098,176.417,26.338,154.390
C06292=1083.466,345.280,-93.132,176.419,26.343,154.391
C06293=1083.473,345.528,-93.167,176.423,26.349,154.392
C06294=1083.479,345.774,-93.201,176.426,26.353,154.393
C06295=1083.484,346.022,-93.236,176.429,26.358,154.393
C06296=1083.490,346.270,-93.271,176.433,26.363,154.394
C06297=1083.496,346.517,-93.305,176.436,26.368,154.395
C06298=1083.502,346.765,-93.340,176.438,26.373,154.396
C06299=1083.508,347.012,-93.374,176.441,26.378,154.397
C06300=1083.514,347.260,-93.409,176.445,26.383,154.397
C06301=1083.520,347.507,-93.444,176.448,26.389,154.398
C06302=1083.526,347.755,-93.479,176.451,26.393,154.399
C06303=1083.532,348.002,-93.514,176.455,26.399,154.400
C06304=1083.538,348.250,-93.548,176.458,26.404,154.401
C06305=1083.544,348.497,-93.584,176.460,26.409,154.402
C06306=1083.550,348.745,-93.618,176.464,26.414,154.402
C06307=1083.555,348.993,-93.653,176.467,26.419,154.403
C06308=1083.562,349.240,-93.688,176.470,26.424,154.404
C06309=1083.567,349.488,-93.723,176.474,26.430,154.405
C06310=1083.574,349.735,-93.758,176.477,26.434,154.406
C06311=1083.579,349.982,-93.793,176.479,26.440,154.407
C06312=1083.586,350.230,-93.827,176.483,26.445,154.408
C06313=1083.591,350.477,-93.863,176.486,26.450,154.408
C06314=1083.598,350.725,-93.897,176.489,26.455,154.409
C06315=1083.604,350.973,-93.933,176.493,26.460,154.410
C06316=1083.610,351.219,-93.968,176.496,26.465,154.411
C06317=1083.616,351.468,-94.003,176.499,26.471,154.412
C06318=1083.622,351.714,-94.038,176.502,26.476,154.413
C06319=1083.628,351.962,-94.073,176.505,26.481,154.414
C06320=1083.634,352.210,-94.108,176.509,26.487,154.414
C06321=1083.640,352.457,-94.143,176.512,26.491,154.415
C06322=1083.646,352.704,-94.179,176.515,26.497,154.416
C06323=1083.653,352.952,-94.214,176.518,26.502,154.417
C06324=1083.658,353.199,-94.249,176.521,26.507,154.418
C06325=1083.664,353.447,-94.284,176.525,26.513,154.419
C06326=1083.670,353.694,-94.319,176.528,26.518,154.420
C06327=1083.676,353.941,-94.355,176.531,26.523,154.421
C06328=1083.682,354.189,-94.391,176.534,26.529,154.422
C06329=1083.688,354.436,-94.425,176.537,26.534,154.422
C06330=1083.694,354.683,-94.461,176.541,26.539,154.423
C06331=1083.700,354.931,-94.497,176.544,26.544,154.424
C06332=1083.705,355.179,-94.531,176.547,26.550,154.425
C06333=1083.711,355.426,-94.567,176.550,26.555,154.426
C06334=1083.718,355.674,-94.602,176.553,26.561,154.427
C06335=1083.724,355.921,-94.638,176.557,26.566,154.428
C06336=1083.730,356.168,-94.673,176.560,26.571,154.429
C06337=1083.736,356.416,-94.709,176.563,26.577,154.430
C06338=1083.743,356.663,-94.745,176.566,26.582,154.431
C06339=1083.752,357.069,-94.803,176.572,26.591,154.432
C06340=1083.762,357.474,-94.861,176.576,26.600,154.434
C06341=1083.772,357.880,-94.920,176.582,26.609,154.435
C06342=1083.781,358.286,-94.978,176.588,26.618,154.437
C06343=1083.788,358.533,-95.014,176.590,26.623,154.438
C06344=1083.794,358.781,-95.050,176.594,26.629,154.438
C06345=1083.800,359.028,-95.086,176.597,26.635,154.440
C06346=1083.806,359.275,-95.121,176.601,26.640,154.440
C06347=1083.812,359.522,-95.157,176.603,26.645,154.441
C06348=1083.818,359.770,-95.193,176.607,26.651,154.442
C06349=1083.824,360.018,-95.229,176.610,26.657,154.443
C06350=1083.830,360.265,-95.265,176.614,26.662,154.444
C06351=1083.836,360.512,-95.301,176.617,26.668,154.445
C06352=1083.842,360.759,-95.336,176.620,26.674,154.446
C06353=1083.848,361.006,-95.373,176.623,26.679,154.447
C06354=1083.854,361.254,-95.409,176.627,26.685,154.448
C06355=1083.861,361.501,-95.445,176.630,26.690,154.449
C06356=1083.867,361.749,-95.481,176.633,26.696,154.450
C06357=1083.873,361.997,-95.516,176.636,26.702,154.451
C06358=1083.878,362.243,-95.553,176.640,26.708,154.452
C06359=1083.884,362.491,-95.588,176.643,26.713,154.453
C06360=1083.891,362.738,-95.625,176.646,26.719,154.454
C06361=1083.897,362.985,-95.661,176.649,26.724,154.455
C06362=1083.903,363.232,-95.697,176.653,26.730,154.456
C06363=1083.909,363.479,-95.733,176.656,26.736,154.457
C06364=1083.915,363.727,-95.769,176.659,26.742,154.458
C06365=1083.922,363.974,-95.805,176.662,26.747,154.459
C06366=1083.928,364.222,-95.841,176.666,26.753,154.460
C06367=1083.933,364.469,-95.878,176.669,26.759,154.461
C06368=1083.940,364.716,-95.915,176.672,26.765,154.462
C06369=1083.945,364.963,-95.951,176.675,26.770,154.463
C06370=1083.952,365.210,-95.986,176.679,26.776,154.464
C06371=1083.958,365.457,-96.023,176.682,26.782,154.465
C06372=1083.964,365.704,-96.059,176.685,26.788,154.466
C06373=1083.970,365.952,-96.096,176.689,26.794,154.467
C06374=1083.976,366.199,-96.132,176.692,26.799,154.468
C06375=1083.982,366.446,-96.169,176.695,26.806,154.469
C06376=1083.988,366.694,-96.206,176.698,26.811,154.470
C06377=1083.994,366.941,-96.242,176.702,26.817,154.471
C06378=1084.000,367.188,-96.279,176.705,26.824,154.472
C06379=1084.006,367.435,-96.316,176.708,26.830,154.473
C06380=1084.012,367.682,-96.352,176.711,26.835,154.474
C06381=1084.018,367.930,-96.388,176.715,26.841,154.475
C06382=1084.024,368.177,-96.425,176.718,26.847,154.476
C06383=1084.030,368.424,-96.461,176.721,26.853,154.478
C06384=1084.037,368.672,-96.498,176.725,26.859,154.479
C06385=1084.042,368.919,-96.535,176.728,26.865,154.480
C06386=1084.049,369.166,-96.571,176.731,26.871,154.481
C06387=1084.055,369.412,-96.608,176.735,26.877,154.482
C06388=1084.061,369.660,-96.645,176.738,26.883,154.483
C06389=1084.067,369.907,-96.682,176.741,26.890,154.484
C06390=1084.073,370.154,-96.719,176.744,26.895,154.485
C06391=1084.079,370.365,-96.750,176.747,26.901,154.486
C06392=1084.084,370.576,-96.781,176.750,26.906,154.487
C06393=1084.088,370.787,-96.813,176.753,26.911,154.488
C06394=1084.094,370.998,-96.844,176.756,26.916,154.489
C06395=1084.100,371.208,-96.876,176.759,26.921,154.490
C06396=1084.105,371.419,-96.908,176.761,26.927,154.491
C06397=1084.110,371.629,-96.939,176.764,26.932,154.492
C06398=1084.115,371.841,-96.970,176.767,26.937,154.493
C06399=1084.121,372.088,-97.007,176.771,26.944,154.494
C06400=1084.127,372.335,-97.044,176.774,26.949,154.495
C06401=1084.134,372.583,-97.081,176.777,26.956,154.496
C06402=1084.140,372.829,-97.119,176.780,26.962,154.497
C06403=1084.146,373.077,-97.155,176.784,26.968,154.498
C06404=1084.153,373.324,-97.192,176.787,26.974,154.499
C06405=1084.158,373.570,-97.229,176.790,26.980,154.500
C06406=1084.165,373.818,-97.266,176.794,26.987,154.501
C06407=1084.171,374.065,-97.304,176.797,26.993,154.503
C06408=1084.177,374.312,-97.341,176.800,26.999,154.504
C06409=1084.183,374.559,-97.377,176.804,27.006,154.505
C06410=1084.189,374.806,-97.415,176.807,27.012,154.506
C06411=1084.195,375.053,-97.452,176.810,27.018,154.507
C06412=1084.201,375.301,-97.490,176.814,27.025,154.508
C06413=1084.208,375.547,-97.528,176.817,27.031,154.510
C06414=1084.213,375.795,-97.565,176.820,27.038,154.511
C06415=1084.219,376.041,-97.602,176.824,27.044,154.512
C06416=1084.226,376.288,-97.639,176.827,27.051,154.513
C06417=1084.232,376.536,-97.677,176.831,27.057,154.514
C06418=1084.238,376.783,-97.715,176.834,27.063,154.516
C06419=1084.244,377.030,-97.752,176.837,27.070,154.517
C06420=1084.250,377.276,-97.789,176.841,27.077,154.518
C06421=1084.257,377.524,-97.827,176.843,27.083,154.519
C06422=1084.263,377.771,-97.865,176.847,27.089,154.520
C06423=1084.268,378.018,-97.902,176.851,27.096,154.521
C06424=1084.276,378.265,-97.939,176.854,27.103,154.523
C06425=1084.282,378.512,-97.977,176.857,27.109,154.524
C06426=1084.287,378.759,-98.015,176.861,27.115,154.525
C06427=1084.294,379.006,-98.053,176.864,27.122,154.526
C06428=1084.300,379.253,-98.090,176.868,27.129,154.528
C06429=1084.306,379.500,-98.127,176.871,27.135,154.529
C06430=1084.313,379.747,-98.165,176.874,27.142,154.530
C06431=1084.319,379.994,-98.203,176.878,27.149,154.531
C06432=1084.324,380.241,-98.241,176.881,27.155,154.532
C06433=1084.331,380.488,-98.279,176.884,27.162,154.534
C06434=1084.337,380.735,-98.317,176.888,27.168,154.535
C06435=1084.344,380.982,-98.354,176.891,27.175,154.536
C06436=1084.350,381.229,-98.392,176.895,27.182,154.537
C06437=1084.356,381.476,-98.430,176.898,27.189,154.539
C06438=1084.362,381.723,-98.468,176.901,27.195,154.540
C06439=1084.368,381.970,-98.506,176.905,27.202,154.541
C06440=1084.375,382.217,-98.544,176.908,27.209,154.542
C06441=1084.381,382.463,-98.582,176.912,27.216,154.544
C06442=1084.388,382.711,-98.620,176.915,27.222,154.545
C06443=1084.393,382.957,-98.658,176.918,27.229,154.546
C06444=1084.399,383.204,-98.696,176.922,27.236,154.548
C06445=1084.406,383.452,-98.734,176.925,27.243,154.549
C06446=1084.412,383.698,-98.772,176.929,27.250,154.550
C06447=1084.417,383.923,-98.807,176.932,27.257,154.552
C06448=1084.424,384.148,-98.842,176.934,27.263,154.553
C06449=1084.429,384.373,-98.877,176.938,27.269,154.554
C06450=1084.435,384.597,-98.911,176.941,27.276,154.555
C06451=1084.440,384.823,-98.946,176.945,27.282,154.556
C06452=1084.446,385.048,-98.982,176.947,27.289,154.558
C06453=1084.452,385.273,-99.016,176.951,27.295,154.559
C06454=1084.457,385.497,-99.051,176.954,27.301,154.560
C06455=1084.463,385.745,-99.089,176.957,27.309,154.561
C06456=1084.470,385.991,-99.128,176.961,27.315,154.563
C06457=1084.476,386.238,-99.166,176.964,27.322,154.564
C06458=1084.482,386.485,-99.204,176.967,27.330,154.565
C06459=1084.488,386.732,-99.243,176.971,27.336,154.567
C06460=1084.494,386.978,-99.282,176.974,27.344,154.568
C06461=1084.501,387.226,-99.320,176.978,27.351,154.569
C06462=1084.508,387.473,-99.359,176.981,27.358,154.571
C06463=1084.514,387.719,-99.396,176.985,27.366,154.572
C06464=1084.520,387.967,-99.436,176.988,27.372,154.573
C06465=1084.526,388.213,-99.474,176.992,27.380,154.575
C06466=1084.532,388.460,-99.512,176.995,27.387,154.576
C06467=1084.539,388.707,-99.551,176.998,27.394,154.578
C06468=1084.545,388.953,-99.590,177.002,27.401,154.579
C06469=1084.551,389.201,-99.628,177.005,27.409,154.580
C06470=1084.558,389.448,-99.667,177.009,27.416,154.582
C06471=1084.564,389.694,-99.706,177.012,27.423,154.583
C06472=1084.571,389.941,-99.744,177.016,27.430,154.585
C06473=1084.576,390.187,-99.784,177.019,27.438,154.586
C06474=1084.583,390.435,-99.822,177.023,27.445,154.587
C06475=1084.590,390.681,-99.861,177.026,27.452,154.589
C06476=1084.596,390.928,-99.900,177.030,27.460,154.590
C06477=1084.602,391.175,-99.938,177.033,27.467,154.592
C06478=1084.609,391.421,-99.977,177.037,27.475,154.593
C06479=1084.615,391.669,-100.017,177.040,27.482,154.595
C06480=1084.622,391.915,-100.056,177.044,27.490,154.596
C06481=1084.628,392.162,-100.094,177.048,27.497,154.598
C06482=1084.634,392.409,-100.133,177.051,27.505,154.599
C06483=1084.641,392.655,-100.172,177.055,27.512,154.600
C06484=1084.647,392.903,-100.212,177.058,27.520,154.602
C06485=1084.653,393.149,-100.250,177.062,27.528,154.603
C06486=1084.659,393.396,-100.290,177.065,27.535,154.605
C06487=1084.666,393.643,-100.328,177.069,27.543,154.606
C06488=1084.672,393.890,-100.368,177.072,27.551,154.608
C06489=1084.678,394.137,-100.407,177.076,27.558,154.609
C06490=1084.685,394.383,-100.447,177.079,27.566,154.611
C06491=1084.691,394.630,-100.486,177.083,27.574,154.612
C06492=1084.698,394.876,-100.525,177.086,27.581,154.614
C06493=1084.704,395.124,-100.564,177.090,27.589,154.615
C06494=1084.710,395.370,-100.604,177.093,27.597,154.617
C06495=1084.717,395.617,-100.643,177.097,27.605,154.619
C06496=1084.723,395.864,-100.683,177.100,27.612,154.620
C06497=1084.729,396.111,-100.722,177.104,27.620,154.622
C06498=1084.735,396.357,-100.761,177.107,27.628,154.623
C06499=1084.742,396.604,-100.801,177.111,27.636,154.625
C06500=1084.748,396.850,-100.841,177.114,27.644,154.626
C06501=1084.755,397.097,-100.880,177.118,27.652,154.628
C06502=1084.761,397.344,-100.919,177.121,27.660,154.629
C06503=1084.767,397.575,-100.957,177.125,27.667,154.631
C06504=1084.773,397.807,-100.994,177.128,27.675,154.632
C06505=1084.779,398.038,-101.031,177.131,27.682,154.634
C06506=1084.785,398.270,-101.068,177.134,27.690,154.635
C06507=1084.791,398.502,-101.105,177.138,27.697,154.637
C06508=1084.797,398.733,-101.143,177.141,27.705,154.638
C06509=1084.803,398.964,-101.180,177.145,27.712,154.640
C06510=1084.809,399.196,-101.217,177.148,27.720,154.641
C06511=1084.815,399.444,-101.257,177.151,27.728,154.643
C06512=1084.821,399.691,-101.297,177.155,27.737,154.645
C06513=1084.828,399.938,-101.337,177.159,27.745,154.646
C06514=1084.835,400.186,-101.377,177.162,27.753,154.648
C06515=1084.841,400.433,-101.417,177.166,27.761,154.650
C06516=1084.848,400.679,-101.457,177.169,27.769,154.651
C06517=1084.854,400.926,-101.497,177.173,27.778,154.653
C06518=1084.860,401.173,-101.537,177.176,27.786,154.655
C06519=1084.866,401.419,-101.577,177.181,27.795,154.656
C06520=1084.873,401.666,-101.617,177.184,27.803,154.658
C06521=1084.879,401.912,-101.657,177.187,27.811,154.660
C06522=1084.886,402.159,-101.697,177.191,27.819,154.661
C06523=1084.893,402.406,-101.738,177.194,27.828,154.663
C06524=1084.899,402.653,-101.778,177.198,27.836,154.665
C06525=1084.905,402.899,-101.818,177.202,27.845,154.667
C06526=1084.912,403.146,-101.858,177.206,27.853,154.668
C06527=1084.918,403.392,-101.898,177.209,27.862,154.670
C06528=1084.925,403.639,-101.939,177.213,27.870,154.672
C06529=1084.931,403.886,-101.979,177.217,27.879,154.673
C06530=1084.938,404.133,-102.019,177.220,27.887,154.675
C06531=1084.944,404.379,-102.059,177.224,27.896,154.677
C06532=1084.951,404.626,-102.100,177.227,27.905,154.679
C06533=1084.958,404.873,-102.140,177.232,27.913,154.680
C06534=1084.964,405.119,-102.180,177.235,27.922,154.682
C06535=1084.970,405.366,-102.221,177.238,27.931,154.684
C06536=1084.976,405.612,-102.262,177.242,27.939,154.686
C06537=1084.983,405.859,-102.302,177.246,27.948,154.687
C06538=1084.990,406.106,-102.343,177.250,27.957,154.689
C06539=1084.996,406.352,-102.383,177.253,27.966,154.691
C06540=1085.002,406.598,-102.424,177.256,27.974,154.693
C06541=1085.009,406.846,-102.465,177.261,27.984,154.695
C06542=1085.015,407.092,-102.505,177.264,27.992,154.696
C06543=1085.022,407.338,-102.546,177.268,28.001,154.698
C06544=1085.028,407.586,-102.587,177.272,28.010,154.700
C06545=1085.035,407.831,-102.628,177.275,28.019,154.702
C06546=1085.041,408.078,-102.668,177.279,28.028,154.704
C06547=1085.048,408.325,-102.710,177.283,28.037,154.706
C06548=1085.054,408.571,-102.750,177.287,28.046,154.707
C06549=1085.060,408.818,-102.791,177.291,28.056,154.709
C06550=1085.067,409.065,-102.832,177.294,28.065,154.711
C06551=1085.073,409.311,-102.873,177.298,28.073,154.713
C06552=1085.080,409.558,-102.914,177.302,28.083,154.715
C06553=1085.087,409.804,-102.955,177.305,28.092,154.717
C06554=1085.093,410.050,-102.996,177.309,28.101,154.719
C06555=1085.100,410.298,-103.037,177.313,28.111,154.721
C06556=1085.106,410.544,-103.078,177.317,28.119,154.723
C06557=1085.113,410.790,-103.119,177.321,28.129,154.725
C06558=1085.119,411.037,-103.161,177.324,28.139,154.727
C06559=1085.125,411.270,-103.199,177.328,28.147,154.728
C06560=1085.131,411.502,-103.238,177.331,28.156,154.730
C06561=1085.138,411.735,-103.277,177.336,28.165,154.732
C06562=1085.144,411.968,-103.316,177.339,28.174,154.734
C06563=1085.150,412.200,-103.355,177.342,28.183,154.736
C06564=1085.156,412.433,-103.394,177.346,28.191,154.738
C06565=1085.162,412.665,-103.433,177.349,28.201,154.739
C06566=1085.169,412.898,-103.472,177.353,28.209,154.741
C06567=1085.175,413.145,-103.514,177.357,28.219,154.743
C06568=1085.182,413.391,-103.555,177.361,28.228,154.745
C06569=1085.189,413.638,-103.596,177.365,28.238,154.747
C06570=1085.195,413.884,-103.637,177.369,28.248,154.749
C06571=1085.202,414.131,-103.679,177.373,28.257,154.751
C06572=1085.209,414.377,-103.720,177.377,28.267,154.753
C06573=1085.215,414.623,-103.762,177.380,28.277,154.755
C06574=1085.222,414.870,-103.803,177.385,28.287,154.757
C06575=1085.229,415.116,-103.846,177.388,28.296,154.759
C06576=1085.235,415.362,-103.887,177.392,28.306,154.762
C06577=1085.242,415.609,-103.928,177.396,28.316,154.764
C06578=1085.249,415.856,-103.970,177.400,28.326,154.766
C06579=1085.255,416.102,-104.012,177.404,28.336,154.768
C06580=1085.263,416.348,-104.054,177.408,28.346,154.770
C06581=1085.269,416.595,-104.095,177.412,28.356,154.772
C06582=1085.275,416.841,-104.138,177.416,28.366,154.774
C06583=1085.282,417.088,-104.179,177.420,28.376,154.776
C06584=1085.288,417.334,-104.221,177.424,28.386,154.778
C06585=1085.295,417.580,-104.263,177.427,28.396,154.780
C06586=1085.302,417.827,-104.305,177.431,28.406,154.783
C06587=1085.309,418.073,-104.347,177.436,28.416,154.785
C06588=1085.316,418.319,-104.390,177.439,28.426,154.787
C06589=1085.322,418.565,-104.431,177.443,28.437,154.789
C06590=1085.329,418.812,-104.474,177.448,28.447,154.791
C06591=1085.335,419.059,-104.515,177.452,28.457,154.793
C06592=1085.342,419.305,-104.558,177.455,28.467,154.796
C06593=1085.348,419.550,-104.600,177.460,28.478,154.798
C06594=1085.355,419.797,-104.642,177.464,28.488,154.800
C06595=1085.362,420.044,-104.685,177.467,28.499,154.802
C06596=1085.369,420.290,-104.727,177.471,28.509,154.804
C06597=1085.376,420.536,-104.769,177.476,28.520,154.807
C06598=1085.383,420.782,-104.812,177.480,28.530,154.809
C06599=1085.389,421.029,-104.853,177.483,28.541,154.811
C06600=1085.396,421.275,-104.896,177.488,28.551,154.813
C06601=1085.403,421.521,-104.938,177.492,28.562,154.816
C06602=1085.409,421.767,-104.981,177.496,28.572,154.818
C06603=1085.416,422.014,-105.023,177.501,28.583,154.820
C06604=1085.423,422.260,-105.066,177.504,28.593,154.822
C06605=1085.430,422.506,-105.108,177.508,28.604,154.825
C06606=1085.436,422.753,-105.151,177.512,28.615,154.827
C06607=1085.443,422.999,-105.194,177.517,28.626,154.829
C06608=1085.450,423.245,-105.236,177.521,28.637,154.832
C06609=1085.457,423.492,-105.279,177.525,28.648,154.834
C06610=1085.464,423.737,-105.322,177.528,28.659,154.836
C06611=1085.471,423.983,-105.365,177.533,28.669,154.839
C06612=1085.477,424.230,-105.408,177.537,28.681,154.841
C06613=1085.484,424.476,-105.450,177.541,28.692,154.844
C06614=1085.491,424.722,-105.494,177.546,28.703,154.846
C06615=1085.497,424.962,-105.535,177.550,28.714,154.848
C06616=1085.504,425.203,-105.577,177.554,28.725,154.851
C06617=1085.510,425.443,-105.619,177.557,28.736,154.853
C06618=1085.517,425.684,-105.661,177.562,28.746,154.855
C06619=1085.524,425.925,-105.703,177.566,28.758,154.858
C06620=1085.530,426.165,-105.746,177.570,28.768,154.860
C06621=1085.537,426.406,-105.788,177.575,28.779,154.863
C06622=1085.544,426.647,-105.830,177.578,28.790,154.865
C06623=1085.551,426.893,-105.873,177.582,28.802,154.867
C06624=1085.557,427.139,-105.916,177.586,28.813,154.870
C06625=1085.565,427.385,-105.959,177.591,28.825,154.872
C06626=1085.572,427.630,-106.002,177.595,28.836,154.875
C06627=1085.578,427.877,-106.046,177.599,28.847,154.877
C06628=1085.586,428.123,-106.089,177.604,28.859,154.880
C06629=1085.592,428.369,-106.133,177.608,28.871,154.882
C06630=1085.599,428.615,-106.176,177.612,28.882,154.885
C06631=1085.606,428.861,-106.219,177.616,28.894,154.888
C06632=1085.613,429.107,-106.263,177.621,28.906,154.890
C06633=1085.620,429.353,-106.306,177.626,28.918,154.893
C06634=1085.627,429.599,-106.350,177.630,28.929,154.895
C06635=1085.634,429.845,-106.393,177.634,28.941,154.898
C06636=1085.640,430.091,-106.437,177.639,28.953,154.900
C06637=1085.647,430.337,-106.481,177.643,28.965,154.903
C06638=1085.655,430.583,-106.525,177.647,28.977,154.906
C06639=1085.661,430.829,-106.569,177.651,28.989,154.908
C06640=1085.668,431.075,-106.612,177.655,29.001,154.911
C06641=1085.675,431.322,-106.656,177.660,29.013,154.914
C06642=1085.682,431.567,-106.699,177.664,29.025,154.916
C06643=1085.689,431.813,-106.743,177.669,29.037,154.919
C06644=1085.696,432.060,-106.787,177.674,29.049,154.922
C06645=1085.703,432.305,-106.831,177.678,29.062,154.924
C06646=1085.710,432.551,-106.875,177.682,29.074,154.927
C06647=1085.717,432.797,-106.919,177.686,29.086,154.930
C06648=1085.724,433.043,-106.963,177.691,29.099,154.933
C06649=1085.731,433.289,-107.007,177.696,29.111,154.935
C06650=1085.738,433.535,-107.052,177.700,29.124,154.938
C06651=1085.744,433.781,-107.096,177.704,29.136,154.941
C06652=1085.751,434.026,-107.139,177.708,29.149,154.944
C06653=1085.759,434.272,-107.184,177.714,29.161,154.947
C06654=1085.765,434.518,-107.228,177.718,29.174,154.949
C06655=1085.773,434.765,-107.273,177.722,29.187,154.952
C06656=1085.779,435.011,-107.317,177.726,29.199,154.955
C06657=1085.786,435.257,-107.362,177.732,29.212,154.958
C06658=1085.794,435.502,-107.406,177.736,29.225,154.961
C06659=1085.801,435.748,-107.450,177.740,29.237,154.963
C06660=1085.808,435.994,-107.495,177.745,29.251,154.966
C06661=1085.815,436.240,-107.540,177.749,29.264,154.969
C06662=1085.822,436.485,-107.584,177.754,29.277,154.972
C06663=1085.829,436.732,-107.628,177.759,29.289,154.975
C06664=1085.835,436.977,-107.673,177.763,29.302,154.978
C06665=1085.843,437.223,-107.718,177.767,29.315,154.981
C06666=1085.849,437.468,-107.762,177.773,29.329,154.984
C06667=1085.857,437.714,-107.807,177.777,29.342,154.987
C06668=1085.865,437.960,-107.852,177.781,29.355,154.990
C06669=1085.872,438.206,-107.896,177.786,29.368,154.993
C06670=1085.879,438.452,-107.941,177.791,29.382,154.996
C06671=1085.885,438.667,-107.981,177.795,29.394,154.999
C06672=1085.891,438.884,-108.020,177.800,29.405,155.001
C06673=1085.898,439.100,-108.060,177.803,29.417,155.004
C06674=1085.903,439.316,-108.099,177.807,29.429,155.006
C06675=1085.910,439.533,-108.139,177.812,29.441,155.009
C06676=1085.917,439.749,-108.179,177.815,29.453,155.012
C06677=1085.923,439.965,-108.218,177.820,29.465,155.015
C06678=1085.929,440.181,-108.258,177.824,29.477,155.017
C06679=1085.937,440.427,-108.303,177.829,29.491,155.020
C06680=1085.944,440.673,-108.349,177.834,29.504,155.023
C06681=1085.951,440.919,-108.394,177.838,29.518,155.027
C06682=1085.958,441.164,-108.438,177.843,29.532,155.030
C06683=1085.965,441.409,-108.484,177.848,29.546,155.033
C06684=1085.973,441.655,-108.529,177.853,29.560,155.036
C06685=1085.979,441.901,-108.575,177.857,29.574,155.039
C06686=1085.987,442.147,-108.620,177.862,29.588,155.042
C06687=1085.994,442.392,-108.665,177.867,29.602,155.046
C06688=1086.001,442.637,-108.711,177.872,29.616,155.049
C06689=1086.008,442.884,-108.757,177.877,29.631,155.052
C06690=1086.016,443.129,-108.802,177.881,29.645,155.055
C06691=1086.023,443.375,-108.848,177.887,29.659,155.059
C06692=1086.030,443.620,-108.894,177.891,29.673,155.062
C06693=1086.038,443.866,-108.940,177.896,29.688,155.065
C06694=1086.045,444.112,-108.985,177.901,29.703,155.069
C06695=1086.052,444.357,-109.031,177.906,29.717,155.072
C06696=1086.059,444.602,-109.076,177.911,29.731,155.075
C06697=1086.067,444.848,-109.122,177.916,29.746,155.079
C06698=1086.074,445.094,-109.168,177.920,29.761,155.082
C06699=1086.081,445.339,-109.214,177.926,29.776,155.086
C06700=1086.088,445.585,-109.260,177.930,29.790,155.089
C06701=1086.096,445.830,-109.306,177.934,29.805,155.092
C06702=1086.103,446.075,-109.353,177.939,29.819,155.096
C06703=1086.111,446.321,-109.398,177.942,29.834,155.099
C06704=1086.118,446.567,-109.445,177.945,29.849,155.103
C06705=1086.126,446.813,-109.490,177.949,29.863,155.106
C06706=1086.133,447.058,-109.537,177.952,29.878,155.110
C06707=1086.140,447.303,-109.584,177.955,29.892,155.113
C06708=1086.148,447.549,-109.629,177.958,29.907,155.117
C06709=1086.155,447.795,-109.676,177.960,29.921,155.120
C06710=1086.162,448.039,-109.722,177.962,29.936,155.124
C06711=1086.169,448.285,-109.768,177.965,29.951,155.127
C06712=1086.178,448.531,-109.814,177.967,29.966,155.131
C06713=1086.185,448.776,-109.861,177.969,29.980,155.134
C06714=1086.192,449.022,-109.907,177.971,29.994,155.138
C06715=1086.200,449.267,-109.954,177.973,30.009,155.142
C06716=1086.208,449.512,-110.000,177.974,30.023,155.145
C06717=1086.217,449.758,-110.046,177.975,30.037,155.149
C06718=1086.228,450.004,-110.090,177.976,30.050,155.152
C06719=1085.852,449.996,-110.294,177.941,30.235,155.202
C06720=1085.841,449.749,-110.249,177.939,30.222,155.199
C06721=1085.831,449.504,-110.202,177.938,30.208,155.195
C06722=1085.823,449.259,-110.156,177.936,30.194,155.192
C06723=1085.817,449.015,-110.110,177.935,30.179,155.188
C06724=1085.808,448.768,-110.063,177.933,30.165,155.184
C06725=1085.801,448.523,-110.017,177.930,30.150,155.181
C06726=1085.794,448.278,-109.971,177.928,30.136,155.177
C06727=1085.786,448.033,-109.924,177.926,30.121,155.174
C06728=1085.779,447.786,-109.877,177.924,30.106,155.170
C06729=1085.771,447.541,-109.832,177.920,30.092,155.167
C06730=1085.764,447.296,-109.785,177.918,30.077,155.163
C06731=1085.756,447.050,-109.739,177.914,30.063,155.160
C06732=1085.749,446.805,-109.692,177.911,30.048,155.156
C06733=1085.742,446.559,-109.646,177.908,30.033,155.153
C06734=1085.735,446.314,-109.600,177.904,30.019,155.149
C06735=1085.728,446.068,-109.554,177.901,30.004,155.146
C06736=1085.719,445.823,-109.507,177.896,29.990,155.142
C06737=1085.712,445.577,-109.461,177.892,29.975,155.139
C06738=1085.705,445.332,-109.415,177.887,29.960,155.135
C06739=1085.698,445.086,-109.369,177.882,29.945,155.132
C06740=1085.690,444.840,-109.323,177.878,29.930,155.128
C06741=1085.683,444.595,-109.278,177.872,29.916,155.125
C06742=1085.676,444.349,-109.232,177.867,29.901,155.122
C06743=1085.668,444.104,-109.186,177.863,29.887,155.118
C06744=1085.661,443.858,-109.140,177.857,29.872,155.115
C06745=1085.653,443.613,-109.094,177.852,29.857,155.112
C06746=1085.646,443.367,-109.048,177.848,29.843,155.108
C06747=1085.640,443.122,-109.003,177.842,29.829,155.105
C06748=1085.632,442.877,-108.957,177.837,29.815,155.102
C06749=1085.625,442.631,-108.912,177.832,29.800,155.099
C06750=1085.618,442.385,-108.866,177.827,29.786,155.095
C06751=1085.610,442.139,-108.820,177.823,29.772,155.092
C06752=1085.603,441.893,-108.775,177.817,29.758,155.089
C06753=1085.595,441.648,-108.729,177.813,29.744,155.086
C06754=1085.588,441.402,-108.683,177.808,29.730,155.083
C06755=1085.581,441.157,-108.639,177.803,29.716,155.079
C06756=1085.574,440.911,-108.593,177.798,29.702,155.076
C06757=1085.566,440.665,-108.548,177.794,29.688,155.073
C06758=1085.559,440.419,-108.503,177.788,29.674,155.070
C06759=1085.551,440.174,-108.458,177.784,29.661,155.067
C06760=1085.546,439.965,-108.419,177.779,29.649,155.064
C06761=1085.540,439.756,-108.381,177.776,29.637,155.061
C06762=1085.534,439.547,-108.343,177.771,29.626,155.059
C06763=1085.528,439.338,-108.303,177.768,29.614,155.056
C06764=1085.522,439.129,-108.265,177.763,29.603,155.054
C06765=1085.515,438.920,-108.227,177.760,29.591,155.051
C06766=1085.509,438.711,-108.189,177.755,29.580,155.049
C06767=1085.502,438.502,-108.151,177.751,29.568,155.046
C06768=1085.496,438.256,-108.107,177.746,29.555,155.043
C06769=1085.488,438.010,-108.062,177.742,29.542,155.040
C06770=1085.481,437.764,-108.017,177.737,29.529,155.037
C06771=1085.474,437.519,-107.972,177.732,29.516,155.034
C06772=1085.467,437.273,-107.927,177.728,29.502,155.031
C06773=1085.460,437.027,-107.882,177.722,29.489,155.028
C06774=1085.453,436.781,-107.838,177.718,29.476,155.025
C06775=1085.446,436.535,-107.793,177.714,29.463,155.022
C06776=1085.439,436.290,-107.748,177.709,29.450,155.019
C06777=1085.431,436.044,-107.703,177.704,29.437,155.016
C06778=1085.424,435.798,-107.658,177.700,29.424,155.014
C06779=1085.417,435.552,-107.615,177.695,29.411,155.011
C06780=1085.410,435.306,-107.570,177.690,29.398,155.008
C06781=1085.403,435.061,-107.526,177.686,29.385,155.005
C06782=1085.396,434.814,-107.481,177.681,29.373,155.002
C06783=1085.389,434.569,-107.437,177.677,29.360,154.999
C06784=1085.382,434.323,-107.392,177.672,29.347,154.996
C06785=1085.375,434.077,-107.348,177.667,29.335,154.994
C06786=1085.368,433.832,-107.304,177.663,29.322,154.991
C06787=1085.361,433.585,-107.260,177.659,29.310,154.988
C06788=1085.354,433.340,-107.215,177.653,29.297,154.985
C06789=1085.347,433.093,-107.171,177.649,29.285,154.983
C06790=1085.340,432.848,-107.126,177.645,29.272,154.980
C06791=1085.333,432.602,-107.083,177.641,29.260,154.977
C06792=1085.326,432.355,-107.039,177.636,29.247,154.974
C06793=1085.320,432.110,-106.994,177.632,29.235,154.972
C06794=1085.312,431.864,-106.951,177.627,29.223,154.969
C06795=1085.305,431.618,-106.907,177.622,29.211,154.966
C06796=1085.298,431.372,-106.864,177.618,29.199,154.964
C06797=1085.291,431.126,-106.819,177.614,29.187,154.961
C06798=1085.284,430.880,-106.775,177.609,29.175,154.958
C06799=1085.277,430.634,-106.732,177.605,29.163,154.955
C06800=1085.271,430.388,-106.688,177.601,29.151,154.953
C06801=1085.263,430.142,-106.644,177.596,29.139,154.950
C06802=1085.257,429.896,-106.600,177.592,29.127,154.948
C06803=1085.249,429.650,-106.557,177.587,29.115,154.945
C06804=1085.242,429.404,-106.513,177.582,29.103,154.942
C06805=1085.235,429.158,-106.470,177.578,29.091,154.940
C06806=1085.229,428.912,-106.426,177.574,29.079,154.937
C06807=1085.222,428.666,-106.383,177.569,29.068,154.935
C06808=1085.215,428.420,-106.339,177.565,29.056,154.932
C06809=1085.208,428.173,-106.296,177.561,29.044,154.930
C06810=1085.201,427.927,-106.252,177.556,29.033,154.927
C06811=1085.194,427.682,-106.209,177.552,29.021,154.924
C06812=1085.187,427.435,-106.166,177.548,29.010,154.922
C06813=1085.180,427.189,-106.122,177.543,28.998,154.920
C06814=1085.173,426.943,-106.079,177.539,28.987,154.917
C06815=1085.166,426.697,-106.036,177.535,28.975,154.915
C06816=1085.159,426.456,-105.994,177.531,28.964,154.912
C06817=1085.153,426.215,-105.951,177.527,28.953,154.910
C06818=1085.146,425.974,-105.909,177.522,28.943,154.907
C06819=1085.139,425.732,-105.867,177.518,28.931,154.905
C06820=1085.133,425.491,-105.824,177.514,28.920,154.903
C06821=1085.126,425.250,-105.782,177.509,28.909,154.900
C06822=1085.119,425.009,-105.740,177.506,28.898,154.898
C06823=1085.112,424.768,-105.698,177.502,28.888,154.895
C06824=1085.106,424.521,-105.655,177.497,28.876,154.893
C06825=1085.099,424.276,-105.612,177.493,28.865,154.891
C06826=1085.092,424.030,-105.569,177.489,28.854,154.888
C06827=1085.085,423.783,-105.527,177.484,28.843,154.886
C06828=1085.079,423.537,-105.484,177.481,28.832,154.883
C06829=1085.072,423.291,-105.440,177.477,28.822,154.881
C06830=1085.065,423.045,-105.398,177.472,28.810,154.879
C06831=1085.058,422.798,-105.355,177.468,28.800,154.876
C06832=1085.051,422.552,-105.313,177.464,28.789,154.874
C06833=1085.045,422.306,-105.270,177.459,28.778,154.872
C06834=1085.039,422.059,-105.227,177.456,28.768,154.870
C06835=1085.032,421.813,-105.185,177.451,28.757,154.867
C06836=1085.025,421.567,-105.142,177.447,28.746,154.865
C06837=1085.018,421.320,-105.100,177.443,28.735,154.863
C06838=1085.010,421.074,-105.058,177.439,28.725,154.860
C06839=1085.004,420.829,-105.015,177.435,28.714,154.858
C06840=1084.997,420.583,-104.973,177.431,28.704,154.856
C06841=1084.990,420.336,-104.930,177.426,28.693,154.854
C06842=1084.984,420.090,-104.888,177.423,28.683,154.851
C06843=1084.977,419.844,-104.845,177.419,28.672,154.849
C06844=1084.970,419.597,-104.803,177.414,28.662,154.847
C06845=1084.963,419.350,-104.761,177.410,28.651,154.845
C06846=1084.956,419.104,-104.718,177.406,28.641,154.843
C06847=1084.950,418.858,-104.677,177.402,28.631,154.840
C06848=1084.944,418.612,-104.634,177.398,28.621,154.838
C06849=1084.937,418.365,-104.592,177.394,28.611,154.836
C06850=1084.930,418.119,-104.550,177.390,28.600,154.834
C06851=1084.923,417.873,-104.508,177.386,28.590,154.832
C06852=1084.917,417.626,-104.467,177.382,28.580,154.830
C06853=1084.910,417.380,-104.424,177.378,28.569,154.827
C06854=1084.903,417.134,-104.382,177.374,28.559,154.825
C06855=1084.897,416.888,-104.340,177.370,28.550,154.823
C06856=1084.890,416.641,-104.298,177.366,28.539,154.821
C06857=1084.884,416.394,-104.256,177.362,28.530,154.819
C06858=1084.877,416.149,-104.215,177.358,28.519,154.817
C06859=1084.870,415.902,-104.172,177.354,28.509,154.815
C06860=1084.864,415.655,-104.130,177.350,28.499,154.813
C06861=1084.856,415.409,-104.089,177.346,28.489,154.811
C06862=1084.850,415.163,-104.048,177.342,28.480,154.808
C06863=1084.843,414.916,-104.005,177.338,28.470,154.806
C06864=1084.836,414.670,-103.964,177.335,28.460,154.804
C06865=1084.830,414.423,-103.923,177.330,28.450,154.802
C06866=1084.823,414.177,-103.881,177.327,28.441,154.800
C06867=1084.816,413.930,-103.840,177.322,28.431,154.798
C06868=1084.810,413.684,-103.797,177.318,28.422,154.796
C06869=1084.803,413.438,-103.756,177.315,28.412,154.794
C06870=1084.797,413.192,-103.715,177.310,28.402,154.792
C06871=1084.790,412.945,-103.673,177.307,28.393,154.790
C06872=1084.783,412.712,-103.635,177.303,28.384,154.788
C06873=1084.778,412.478,-103.595,177.300,28.375,154.787
C06874=1084.771,412.246,-103.556,177.295,28.366,154.785
C06875=1084.764,412.011,-103.517,177.292,28.357,154.783
C06876=1084.758,411.778,-103.477,177.288,28.348,154.781
C06877=1084.752,411.545,-103.439,177.285,28.339,154.779
C06878=1084.746,411.312,-103.399,177.281,28.330,154.777
C06879=1084.739,411.079,-103.361,177.278,28.321,154.775
C06880=1084.733,410.833,-103.319,177.273,28.312,154.773
C06881=1084.726,410.586,-103.278,177.270,28.303,154.772
C06882=1084.720,410.339,-103.237,177.265,28.293,154.770
C06883=1084.713,410.092,-103.196,177.262,28.284,154.768
C06884=1084.707,409.846,-103.155,177.259,28.275,154.766
C06885=1084.700,409.599,-103.114,177.254,28.265,154.764
C06886=1084.694,409.353,-103.073,177.251,28.256,154.762
C06887=1084.687,409.106,-103.032,177.246,28.247,154.760
C06888=1084.681,408.859,-102.991,177.243,28.238,154.758
C06889=1084.675,408.614,-102.950,177.239,28.229,154.756
C06890=1084.667,408.367,-102.909,177.235,28.220,154.754
C06891=1084.662,408.120,-102.868,177.232,28.211,154.753
C06892=1084.655,407.874,-102.827,177.228,28.202,154.751
C06893=1084.649,407.627,-102.786,177.224,28.193,154.749
C06894=1084.642,407.381,-102.745,177.220,28.183,154.747
C06895=1084.636,407.134,-102.705,177.217,28.175,154.745
C06896=1084.629,406.887,-102.665,177.212,28.166,154.743
C06897=1084.623,406.641,-102.623,177.209,28.157,154.742
C06898=1084.616,406.394,-102.583,177.206,28.148,154.740
C06899=1084.609,406.147,-102.542,177.202,28.139,154.738
C06900=1084.603,405.901,-102.502,177.198,28.130,154.736
C06901=1084.597,405.654,-102.461,177.194,28.121,154.734
C06902=1084.590,405.407,-102.420,177.191,28.113,154.732
C06903=1084.583,405.161,-102.379,177.187,28.104,154.731
C06904=1084.577,404.915,-102.339,177.183,28.095,154.729
C06905=1084.571,404.668,-102.299,177.179,28.087,154.727
C06906=1084.564,404.421,-102.259,177.176,28.078,154.725
C06907=1084.558,404.174,-102.218,177.172,28.069,154.724
C06908=1084.552,403.928,-102.178,177.168,28.061,154.722
C06909=1084.545,403.681,-102.138,177.164,28.052,154.720
C06910=1084.538,403.435,-102.096,177.161,28.044,154.718
C06911=1084.532,403.188,-102.056,177.157,28.035,154.717
C06912=1084.525,402.942,-102.016,177.154,28.027,154.715
C06913=1084.519,402.695,-101.976,177.149,28.018,154.713
C06914=1084.512,402.449,-101.936,177.146,28.010,154.711
C06915=1084.505,402.201,-101.895,177.142,28.001,154.710
C06916=1084.499,401.954,-101.856,177.139,27.993,154.708
C06917=1084.493,401.708,-101.816,177.135,27.985,154.706
C06918=1084.487,401.461,-101.775,177.132,27.976,154.705
C06919=1084.480,401.215,-101.735,177.127,27.968,154.703
C06920=1084.474,400.968,-101.695,177.124,27.959,154.701
C06921=1084.468,400.722,-101.655,177.121,27.951,154.700
C06922=1084.461,400.475,-101.615,177.117,27.943,154.698
C06923=1084.454,400.228,-101.576,177.113,27.935,154.696
C06924=1084.447,399.981,-101.536,177.110,27.927,154.695
C06925=1084.441,399.735,-101.495,177.106,27.918,154.693
C06926=1084.435,399.487,-101.456,177.103,27.910,154.691
C06927=1084.429,399.241,-101.416,177.099,27.901,154.690
C06928=1084.422,399.009,-101.378,177.096,27.894,154.688
C06929=1084.417,398.777,-101.340,177.092,27.887,154.687
C06930=1084.411,398.544,-101.303,177.089,27.879,154.685
C06931=1084.405,398.311,-101.266,177.085,27.871,154.684
C06932=1084.398,398.079,-101.229,177.082,27.864,154.682
C06933=1084.392,397.847,-101.191,177.079,27.856,154.681
C06934=1084.386,397.615,-101.154,177.075,27.848,154.679
C06935=1084.380,397.382,-101.117,177.072,27.841,154.678
C06936=1084.374,397.135,-101.077,177.068,27.833,154.676
C06937=1084.368,396.888,-101.037,177.065,27.825,154.675
C06938=1084.361,396.641,-100.997,177.061,27.817,154.673
C06939=1084.354,396.395,-100.958,177.058,27.809,154.671
C06940=1084.348,396.148,-100.918,177.054,27.802,154.670
C06941=1084.342,395.901,-100.879,177.050,27.794,154.668
C06942=1084.336,395.655,-100.840,177.047,27.786,154.667
C06943=1084.329,395.408,-100.800,177.043,27.778,154.665
C06944=1084.323,395.161,-100.761,177.040,27.770,154.664
C06945=1084.316,394.914,-100.722,177.036,27.762,154.662
C06946=1084.310,394.668,-100.682,177.033,27.755,154.661
C06947=1084.304,394.421,-100.642,177.029,27.747,154.659
C06948=1084.297,394.174,-100.604,177.026,27.739,154.658
C06949=1084.291,393.927,-100.564,177.022,27.731,154.656
C06950=1084.285,393.681,-100.526,177.019,27.724,154.655
C06951=1084.279,393.434,-100.485,177.015,27.716,154.653
C06952=1084.272,393.187,-100.447,177.011,27.708,154.651
C06953=1084.266,392.940,-100.407,177.008,27.701,154.650
C06954=1084.259,392.693,-100.368,177.004,27.693,154.649
C06955=1084.253,392.447,-100.329,177.001,27.686,154.647
C06956=1084.247,392.200,-100.290,176.997,27.678,154.646
C06957=1084.240,391.953,-100.251,176.994,27.670,154.644
C06958=1084.234,391.706,-100.212,176.990,27.663,154.643
C06959=1084.228,391.460,-100.173,176.987,27.655,154.641
C06960=1084.221,391.213,-100.134,176.983,27.648,154.640
C06961=1084.215,390.966,-100.095,176.979,27.640,154.638
C06962=1084.208,390.719,-100.057,176.976,27.633,154.637
C06963=1084.202,390.473,-100.018,176.973,27.626,154.635
C06964=1084.195,390.226,-99.979,176.969,27.619,154.634
C06965=1084.189,389.979,-99.941,176.966,27.611,154.633
C06966=1084.183,389.731,-99.901,176.962,27.604,154.631
C06967=1084.177,389.485,-99.863,176.959,27.597,154.630
C06968=1084.170,389.238,-99.824,176.955,27.589,154.628
C06969=1084.163,388.992,-99.785,176.952,27.582,154.627
C06970=1084.158,388.745,-99.747,176.948,27.574,154.626
C06971=1084.151,388.498,-99.708,176.944,27.567,154.624
C06972=1084.144,388.251,-99.669,176.941,27.560,154.623
C06973=1084.138,388.004,-99.631,176.937,27.553,154.621
C06974=1084.132,387.757,-99.592,176.934,27.545,154.620
C06975=1084.126,387.511,-99.553,176.931,27.538,154.619
C06976=1084.120,387.263,-99.515,176.927,27.531,154.617
C06977=1084.113,387.017,-99.476,176.924,27.524,154.616
C06978=1084.107,386.771,-99.438,176.920,27.517,154.614
C06979=1084.101,386.523,-99.399,176.917,27.510,154.613
C06980=1084.095,386.277,-99.361,176.913,27.502,154.612
C06981=1084.088,386.029,-99.323,176.909,27.495,154.610
C06982=1084.082,385.783,-99.284,176.907,27.488,154.609
C06983=1084.075,385.536,-99.246,176.903,27.481,154.608
C06984=1084.070,385.310,-99.211,176.899,27.475,154.607
C06985=1084.064,385.084,-99.175,176.897,27.468,154.605
C06986=1084.059,384.859,-99.141,176.893,27.462,154.604
C06987=1084.053,384.633,-99.106,176.890,27.455,154.603
C06988=1084.047,384.408,-99.071,176.887,27.449,154.602
C06989=1084.041,384.183,-99.036,176.884,27.443,154.600
C06990=1084.036,383.957,-99.001,176.881,27.437,154.599
C06991=1084.031,383.732,-98.966,176.877,27.430,154.598
C06992=1084.024,383.485,-98.927,176.875,27.423,154.597
C06993=1084.018,383.238,-98.890,176.871,27.416,154.595
C06994=1084.012,382.991,-98.852,176.867,27.409,154.594
C06995=1084.006,382.744,-98.814,176.864,27.402,154.593
C06996=1083.999,382.497,-98.775,176.860,27.395,154.592
C06997=1083.993,382.251,-98.737,176.857,27.389,154.590
C06998=1083.986,382.003,-98.699,176.854,27.382,154.589
C06999=1083.981,381.756,-98.661,176.850,27.375,154.588
C07000=1083.975,381.510,-98.624,176.846,27.368,154.586
C07001=1083.968,381.262,-98.585,176.844,27.361,154.585
C07002=1083.962,381.015,-98.548,176.840,27.355,154.584
C07003=1083.955,380.768,-98.510,176.836,27.348,154.583
C07004=1083.949,380.522,-98.472,176.833,27.341,154.581
C07005=1083.943,380.274,-98.434,176.830,27.335,154.580
C07006=1083.937,380.027,-98.397,176.826,27.328,154.579
C07007=1083.931,379.781,-98.359,176.823,27.322,154.578
C07008=1083.924,379.533,-98.321,176.819,27.315,154.576
C07009=1083.918,379.287,-98.284,176.817,27.308,154.575
C07010=1083.912,379.040,-98.246,176.813,27.302,154.574
C07011=1083.905,378.793,-98.208,176.809,27.295,154.573
C07012=1083.899,378.546,-98.170,176.806,27.288,154.571
C07013=1083.893,378.298,-98.132,176.803,27.282,154.570
C07014=1083.887,378.051,-98.095,176.799,27.275,154.569
C07015=1083.881,377.805,-98.058,176.795,27.269,154.568
C07016=1083.874,377.517,-98.014,176.792,27.261,154.566
C07017=1083.866,377.229,-97.970,176.788,27.253,154.565
C07018=1083.859,376.942,-97.926,176.784,27.246,154.564
C07019=1083.851,376.654,-97.882,176.780,27.238,154.562
C07020=1083.845,376.407,-97.845,176.777,27.232,154.561
C07021=1083.840,376.159,-97.808,176.773,27.225,154.560
C07022=1083.833,375.913,-97.771,176.770,27.219,154.559
C07023=1083.827,375.666,-97.733,176.767,27.212,154.557
C07024=1083.821,375.418,-97.695,176.763,27.206,154.556
C07025=1083.815,375.171,-97.658,176.760,27.199,154.555
C07026=1083.809,374.924,-97.621,176.757,27.193,154.554
C07027=1083.803,374.678,-97.583,176.753,27.187,154.553
C07028=1083.797,374.430,-97.546,176.749,27.180,154.552
C07029=1083.790,374.183,-97.509,176.747,27.174,154.550
C07030=1083.785,373.936,-97.472,176.743,27.168,154.549
C07031=1083.779,373.689,-97.434,176.739,27.161,154.548
C07032=1083.772,373.442,-97.398,176.737,27.155,154.547
C07033=1083.766,373.195,-97.359,176.733,27.149,154.546
C07034=1083.759,372.948,-97.323,176.729,27.143,154.545
C07035=1083.754,372.700,-97.286,176.726,27.136,154.544
C07036=1083.747,372.454,-97.249,176.723,27.130,154.542
C07037=1083.741,372.207,-97.212,176.720,27.124,154.541
C07038=1083.735,371.959,-97.175,176.716,27.118,154.540
C07039=1083.728,371.712,-97.138,176.713,27.112,154.539
C07040=1083.719,371.330,-97.081,176.708,27.102,154.537
C07041=1083.709,370.948,-97.024,176.703,27.093,154.536
C07042=1083.700,370.566,-96.967,176.697,27.083,154.534
C07043=1083.690,370.184,-96.910,176.692,27.074,154.532
C07044=1083.684,369.937,-96.873,176.689,27.067,154.531
C07045=1083.678,369.690,-96.836,176.686,27.062,154.530
C07046=1083.672,369.442,-96.799,176.682,27.056,154.529
C07047=1083.666,369.195,-96.763,176.679,27.049,154.528
C07048=1083.660,368.948,-96.726,176.676,27.043,154.527
C07049=1083.654,368.701,-96.689,176.672,27.037,154.526
C07050=1083.648,368.454,-96.653,176.669,27.031,154.525
C07051=1083.642,368.207,-96.616,176.666,27.025,154.524
C07052=1083.636,367.959,-96.579,176.663,27.020,154.523
C07053=1083.630,367.712,-96.543,176.659,27.014,154.522
C07054=1083.623,367.465,-96.506,176.655,27.007,154.520
C07055=1083.618,367.218,-96.469,176.653,27.001,154.519
C07056=1083.611,366.971,-96.433,176.649,26.995,154.518
C07057=1083.605,366.724,-96.397,176.646,26.990,154.517
C07058=1083.599,366.476,-96.360,176.642,26.984,154.516
C07059=1083.593,366.229,-96.323,176.639,26.978,154.515
C07060=1083.587,365.982,-96.287,176.636,26.972,154.514
C07061=1083.581,365.734,-96.250,176.633,26.966,154.513
C07062=1083.575,365.487,-96.214,176.629,26.960,154.512
C07063=1083.569,365.240,-96.177,176.626,26.954,154.511
C07064=1083.562,364.993,-96.141,176.623,26.948,154.510
C07065=1083.556,364.746,-96.105,176.620,26.943,154.509
C07066=1083.551,364.498,-96.068,176.616,26.937,154.508
C07067=1083.544,364.251,-96.032,176.613,26.931,154.507
C07068=1083.538,364.003,-95.996,176.610,26.925,154.506
C07069=1083.532,363.756,-95.960,176.606,26.919,154.505
C07070=1083.526,363.509,-95.923,176.603,26.914,154.504
C07071=1083.520,363.262,-95.888,176.599,26.907,154.503
C07072=1083.514,363.015,-95.851,176.597,26.902,154.502
C07073=1083.508,362.768,-95.815,176.593,26.896,154.501
C07074=1083.502,362.521,-95.779,176.590,26.891,154.500
C07075=1083.495,362.274,-95.743,176.586,26.885,154.499
C07076=1083.489,362.026,-95.707,176.583,26.879,154.498
C07077=1083.483,361.779,-95.671,176.581,26.873,154.497
C07078=1083.477,361.531,-95.635,176.577,26.868,154.496
C07079=1083.471,361.284,-95.598,176.574,26.862,154.495
C07080=1083.465,361.037,-95.563,176.570,26.857,154.494
C07081=1083.459,360.789,-95.527,176.567,26.851,154.493
C07082=1083.453,360.542,-95.490,176.564,26.845,154.492
C07083=1083.447,360.295,-95.455,176.561,26.840,154.491
C07084=1083.440,360.048,-95.419,176.557,26.834,154.490
C07085=1083.434,359.800,-95.383,176.554,26.828,154.489
C07086=1083.429,359.553,-95.348,176.550,26.823,154.488
C07087=1083.423,359.305,-95.312,176.548,26.818,154.487
C07088=1083.417,359.058,-95.275,176.544,26.811,154.486
C07089=1083.411,358.811,-95.240,176.541,26.806,154.485
C07090=1083.404,358.563,-95.204,176.538,26.801,154.484
C07091=1083.399,358.316,-95.169,176.534,26.795,154.483
C07092=1083.388,357.909,-95.109,176.529,26.786,154.482
C07093=1083.378,357.502,-95.051,176.524,26.778,154.480
C07094=1083.368,357.095,-94.992,176.518,26.768,154.479
C07095=1083.358,356.688,-94.934,176.513,26.759,154.477
C07096=1083.352,356.442,-94.898,176.510,26.754,154.476
C07097=1083.346,356.194,-94.862,176.507,26.748,154.475
C07098=1083.340,355.947,-94.827,176.504,26.743,154.475
C07099=1083.335,355.700,-94.791,176.500,26.738,154.474
C07100=1083.328,355.452,-94.756,176.497,26.732,154.473
C07101=1083.322,355.205,-94.720,176.494,26.727,154.472
C07102=1083.317,354.958,-94.685,176.490,26.721,154.471
C07103=1083.311,354.710,-94.649,176.488,26.716,154.470
C07104=1083.304,354.462,-94.614,176.484,26.710,154.469
C07105=1083.299,354.215,-94.580,176.481,26.705,154.468
C07106=1083.293,353.967,-94.544,176.478,26.700,154.467
C07107=1083.287,353.720,-94.508,176.474,26.695,154.466
C07108=1083.280,353.473,-94.473,176.471,26.689,154.465
C07109=1083.274,353.225,-94.438,176.468,26.684,154.464
C07110=1083.268,352.978,-94.402,176.465,26.678,154.464
C07111=1083.262,352.731,-94.367,176.462,26.673,154.463
C07112=1083.256,352.483,-94.332,176.458,26.668,154.462
C07113=1083.250,352.235,-94.296,176.455,26.663,154.461
C07114=1083.244,351.988,-94.262,176.452,26.658,154.460
C07115=1083.238,351.741,-94.226,176.449,26.652,154.459
C07116=1083.232,351.493,-94.192,176.446,26.647,154.458
C07117=1083.226,351.246,-94.156,176.443,26.642,154.457
C07118=1083.220,350.998,-94.121,176.439,26.636,154.457
C07119=1083.214,350.751,-94.086,176.436,26.632,154.456
C07120=1083.208,350.503,-94.051,176.433,26.626,154.455
C07121=1083.202,350.256,-94.016,176.429,26.621,154.454
C07122=1083.196,350.008,-93.981,176.427,26.616,154.453
C07123=1083.190,349.761,-93.946,176.424,26.611,154.452
C07124=1083.184,349.513,-93.912,176.420,26.605,154.451
C07125=1083.178,349.266,-93.876,176.417,26.600,154.451
C07126=1083.172,349.018,-93.842,176.414,26.595,154.450
C07127=1083.166,348.771,-93.806,176.410,26.590,154.449
C07128=1083.160,348.524,-93.772,176.407,26.585,154.448
C07129=1083.154,348.276,-93.736,176.405,26.580,154.447
C07130=1083.148,348.029,-93.702,176.401,26.575,154.446
C07131=1083.142,347.781,-93.666,176.398,26.569,154.445
C07132=1083.136,347.534,-93.632,176.395,26.565,154.445
C07133=1083.130,347.286,-93.597,176.391,26.559,154.444
C07134=1083.124,347.039,-93.563,176.388,26.554,154.443
C07135=1083.118,346.791,-93.528,176.385,26.549,154.442
C07136=1083.113,346.544,-93.493,176.382,26.545,154.441
C07137=1083.106,346.296,-93.458,176.379,26.539,154.440
C07138=1083.101,346.048,-93.424,176.376,26.534,154.440
C07139=1083.094,345.801,-93.389,176.373,26.529,154.439
C07140=1083.088,345.553,-93.355,176.369,26.524,154.438
C07141=1083.083,345.305,-93.320,176.366,26.519,154.437
C07142=1083.077,345.058,-93.286,176.363,26.514,154.436
C07143=1083.071,344.811,-93.251,176.360,26.509,154.436
C07144=1083.061,344.407,-93.195,176.355,26.501,154.434
C07145=1083.052,344.003,-93.138,176.350,26.493,154.433
C07146=1083.041,343.599,-93.082,176.345,26.485,154.432
C07147=1083.031,343.195,-93.026,176.339,26.477,154.430
C07148=1083.026,342.948,-92.992,176.337,26.472,154.430
C07149=1083.019,342.700,-92.957,176.333,26.467,154.429
C07150=1083.014,342.453,-92.923,176.330,26.462,154.428
C07151=1083.008,342.205,-92.888,176.327,26.457,154.427
C07152=1083.002,341.957,-92.854,176.324,26.452,154.426
C07153=1082.996,341.710,-92.820,176.320,26.447,154.426
C07154=1082.989,341.462,-92.786,176.317,26.442,154.425
C07155=1082.983,341.215,-92.752,176.314,26.438,154.424
C07156=1082.978,340.967,-92.718,176.311,26.433,154.423
C07157=1082.972,340.719,-92.683,176.307,26.428,154.422
C07158=1082.966,340.472,-92.649,176.305,26.423,154.422
C07159=1082.960,340.225,-92.615,176.302,26.419,154.421
C07160=1082.954,339.977,-92.580,176.299,26.414,154.420
C07161=1082.948,339.729,-92.547,176.296,26.409,154.419
C07162=1082.942,339.481,-92.513,176.292,26.404,154.419
C07163=1082.936,339.234,-92.479,176.289,26.399,154.418
C07164=1082.930,338.986,-92.444,176.286,26.394,154.417
C07165=1082.924,338.739,-92.410,176.283,26.389,154.416
C07166=1082.919,338.491,-92.377,176.280,26.384,154.416
C07167=1082.913,338.243,-92.342,176.276,26.380,154.415
C07168=1082.907,337.995,-92.308,176.273,26.375,154.414
C07169=1082.900,337.748,-92.274,176.270,26.370,154.413
C07170=1082.895,337.500,-92.241,176.267,26.366,154.413
C07171=1082.888,337.252,-92.207,176.265,26.361,154.412
C07172=1082.882,337.005,-92.173,176.261,26.356,154.411
C07173=1082.877,336.757,-92.139,176.258,26.352,154.410
C07174=1082.871,336.510,-92.105,176.255,26.347,154.410
C07175=1082.865,336.262,-92.071,176.252,26.342,154.409
C07176=1082.859,336.014,-92.037,176.249,26.338,154.408
C07177=1082.853,335.767,-92.003,176.246,26.333,154.407
C07178=1082.848,335.519,-91.970,176.242,26.328,154.407
C07179=1082.840,335.271,-91.936,176.239,26.323,154.406
C07180=1082.835,335.023,-91.903,176.236,26.318,154.405
C07181=1082.829,334.776,-91.869,176.233,26.314,154.405
C07182=1082.823,334.528,-91.836,176.230,26.309,154.404
C07183=1082.818,334.281,-91.801,176.227,26.305,154.403
C07184=1082.812,334.033,-91.768,176.224,26.300,154.402
C07185=1082.806,333.785,-91.734,176.220,26.295,154.402
C07186=1082.799,333.537,-91.701,176.218,26.291,154.401
C07187=1082.793,333.290,-91.667,176.215,26.286,154.400
C07188=1082.788,333.042,-91.634,176.212,26.281,154.399
C07189=1082.782,332.794,-91.600,176.209,26.277,154.399
C07190=1082.776,332.547,-91.566,176.206,26.272,154.398
C07191=1082.770,332.299,-91.533,176.203,26.268,154.397
C07192=1082.765,332.052,-91.500,176.200,26.263,154.397
C07193=1082.759,331.804,-91.466,176.196,26.258,154.396
C07194=1082.753,331.556,-91.432,176.193,26.254,154.395
C07195=1082.746,331.308,-91.400,176.190,26.249,154.394
C07196=1082.737,330.899,-91.344,176.185,26.242,154.393
C07197=1082.726,330.489,-91.290,176.180,26.235,154.392
C07198=1082.717,330.080,-91.234,176.175,26.227,154.391
C07199=1082.706,329.671,-91.180,176.170,26.220,154.390
C07200=1082.701,329.423,-91.147,176.167,26.215,154.389
C07201=1082.694,329.175,-91.114,176.164,26.211,154.389
C07202=1082.688,328.928,-91.080,176.161,26.207,154.388
C07203=1082.682,328.680,-91.047,176.158,26.202,154.387
C07204=1082.677,328.432,-91.014,176.155,26.198,154.387
C07205=1082.670,328.185,-90.981,176.152,26.194,154.386
C07206=1082.664,327.936,-90.947,176.148,26.189,154.385
C07207=1082.658,327.689,-90.915,176.145,26.185,154.385
C07208=1082.652,327.441,-90.881,176.142,26.180,154.384
C07209=1082.646,327.193,-90.848,176.139,26.176,154.383
C07210=1082.640,326.945,-90.815,176.136,26.171,154.383
C07211=1082.634,326.698,-90.782,176.133,26.167,154.382
C07212=1082.628,326.450,-90.750,176.130,26.162,154.381
C07213=1082.622,326.202,-90.716,176.127,26.158,154.381
C07214=1082.616,325.954,-90.684,176.124,26.154,154.380
C07215=1082.611,325.707,-90.650,176.121,26.149,154.379
C07216=1082.605,325.458,-90.618,176.118,26.145,154.379
C07217=1082.599,325.210,-90.585,176.115,26.140,154.378
C07218=1082.593,324.964,-90.553,176.112,26.136,154.377
C07219=1082.587,324.716,-90.520,176.109,26.132,154.377
C07220=1082.581,324.468,-90.486,176.106,26.127,154.376
C07221=1082.575,324.220,-90.454,176.103,26.123,154.375
C07222=1082.570,323.972,-90.421,176.100,26.119,154.375
C07223=1082.564,323.724,-90.388,176.097,26.114,154.374
C07224=1082.557,323.477,-90.356,176.094,26.110,154.373
C07225=1082.552,323.229,-90.322,176.091,26.106,154.373
C07226=1082.546,322.981,-90.290,176.088,26.102,154.372
C07227=1082.539,322.733,-90.257,176.085,26.097,154.372
C07228=1082.534,322.485,-90.224,176.081,26.093,154.371
C07229=1082.528,322.238,-90.192,176.078,26.088,154.370
C07230=1082.522,321.990,-90.160,176.075,26.084,154.370
C07231=1082.517,321.742,-90.126,176.072,26.080,154.369
C07232=1082.511,321.494,-90.094,176.069,26.075,154.368
C07233=1082.504,321.246,-90.062,176.066,26.071,154.368
C07234=1082.499,320.998,-90.028,176.063,26.066,154.367
C07235=1082.493,320.751,-89.997,176.060,26.062,154.366
C07236=1082.487,320.503,-89.964,176.057,26.058,154.366
C07237=1082.482,320.255,-89.931,176.054,26.054,154.365
C07238=1082.476,320.007,-89.899,176.051,26.049,154.364
C07239=1082.470,319.760,-89.867,176.048,26.045,154.364
C07240=1082.464,319.512,-89.834,176.046,26.041,154.363
C07241=1082.459,319.264,-89.801,176.043,26.037,154.362
C07242=1082.452,319.016,-89.769,176.040,26.032,154.362
C07243=1082.447,318.768,-89.737,176.037,26.028,154.361
C07244=1082.441,318.521,-89.704,176.034,26.024,154.361
C07245=1082.435,318.272,-89.672,176.031,26.020,154.360
C07246=1082.429,318.025,-89.639,176.028,26.015,154.359
C07247=1082.424,317.777,-89.607,176.025,26.011,154.359
C07248=1082.414,317.361,-89.552,176.020,26.004,154.358
C07249=1082.404,316.945,-89.499,176.015,25.997,154.357
C07250=1082.395,316.528,-89.444,176.010,25.990,154.355
C07251=1082.385,316.113,-89.390,176.005,25.982,154.354
C07252=1082.379,315.865,-89.358,176.002,25.978,154.354
C07253=1082.374,315.617,-89.326,175.999,25.974,154.353
C07254=1082.369,315.369,-89.294,175.996,25.969,154.353
C07255=1082.362,315.121,-89.261,175.993,25.965,154.352
C07256=1082.356,314.873,-89.229,175.990,25.961,154.351
C07257=1082.351,314.626,-89.198,175.987,25.957,154.351
C07258=1082.345,314.377,-89.166,175.984,25.953,154.350
C07259=1082.339,314.129,-89.133,175.982,25.949,154.350
C07260=1082.333,313.881,-89.101,175.979,25.945,154.349
C07261=1082.327,313.634,-89.070,175.976,25.941,154.348
C07262=1082.321,313.386,-89.038,175.973,25.937,154.348
C07263=1082.315,313.138,-89.006,175.970,25.933,154.347
C07264=1082.309,312.891,-88.974,175.967,25.928,154.347
C07265=1082.303,312.642,-88.942,175.964,25.925,154.346
C07266=1082.297,312.394,-88.911,175.961,25.921,154.346
C07267=1082.291,312.147,-88.879,175.958,25.916,154.345
